LIN {X 61.321,Y 108.503,Z 73.500,A 180.000,B 0.000,C 180.000} C_DIS
LIN {X 61.500,Y 108.424,Z 73.500,A 180.000,B 0.000,C 180.000} C_DIS
LIN {X 61.692,Y 108.338,Z 73.500,A 180.000,B 0.000,C 180.000} C_DIS
LIN {X 61.858,Y 108.262,Z 73.500,A 180.000,B 0.000,C 180.000} C_DIS
LIN {X 62.036,Y 108.167,Z 73.500,A 180.000,B 0.000,C 180.000} C_DIS
LIN {X 62.371,Y 107.980,Z 73.500,A 180.000,B 0.000,C 180.000} C_DIS
LIN {X 62.394,Y 107.967,Z 73.500,A 180.000,B 0.000,C 180.000} C_DIS
LIN {X 62.573,Y 107.855,Z 73.500,A 180.000,B 0.000,C 180.000} C_DIS
LIN {X 62.930,Y 107.612,Z 73.500,A 180.000,B 0.000,C 180.000} C_DIS
LIN {X 63.020,Y 107.548,Z 73.500,A 180.000,B 0.000,C 180.000} C_DIS
LIN {X 63.109,Y 107.478,Z 73.500,A 180.000,B 0.000,C 180.000} C_DIS
LIN {X 63.369,Y 107.265,Z 73.500,A 180.000,B 0.000,C 180.000} C_DIS
LIN {X 63.467,Y 107.185,Z 73.500,A 180.000,B 0.000,C 180.000} C_DIS
LIN {X 63.578,Y 107.086,Z 73.500,A 180.000,B 0.000,C 180.000} C_DIS
LIN {X 63.645,Y 107.021,Z 73.500,A 180.000,B 0.000,C 180.000} C_DIS
LIN {X 63.824,Y 106.847,Z 73.500,A 180.000,B 0.000,C 180.000} C_DIS
LIN {X 63.944,Y 106.729,Z 73.500,A 180.000,B 0.000,C 180.000} C_DIS
LIN {X 64.003,Y 106.669,Z 73.500,A 180.000,B 0.000,C 180.000} C_DIS
LIN {X 64.109,Y 106.550,Z 73.500,A 180.000,B 0.000,C 180.000} C_DIS
LIN {X 64.360,Y 106.256,Z 73.500,A 180.000,B 0.000,C 180.000} C_DIS
LIN {X 64.414,Y 106.193,Z 73.500,A 180.000,B 0.000,C 180.000} C_DIS
LIN {X 64.539,Y 106.026,Z 73.500,A 180.000,B 0.000,C 180.000} C_DIS
LIN {X 64.718,Y 105.776,Z 73.500,A 180.000,B 0.000,C 180.000} C_DIS
LIN {X 64.802,Y 105.656,Z 73.500,A 180.000,B 0.000,C 180.000} C_DIS
LIN {X 64.897,Y 105.507,Z 73.500,A 180.000,B 0.000,C 180.000} C_DIS
LIN {X 65.075,Y 105.203,Z 73.500,A 180.000,B 0.000,C 180.000} C_DIS
LIN {X 65.124,Y 105.120,Z 73.500,A 180.000,B 0.000,C 180.000} C_DIS
LIN {X 65.219,Y 104.941,Z 73.500,A 180.000,B 0.000,C 180.000} C_DIS
LIN {X 65.254,Y 104.866,Z 73.500,A 180.000,B 0.000,C 180.000} C_DIS
LIN {X 65.388,Y 104.584,Z 73.500,A 180.000,B 0.000,C 180.000} C_DIS
LIN {X 65.433,Y 104.488,Z 73.500,A 180.000,B 0.000,C 180.000} C_DIS
LIN {X 65.469,Y 104.405,Z 73.500,A 180.000,B 0.000,C 180.000} C_DIS
LIN {X 65.536,Y 104.226,Z 73.500,A 180.000,B 0.000,C 180.000} C_DIS
LIN {X 65.612,Y 104.022,Z 73.500,A 180.000,B 0.000,C 180.000} C_DIS
LIN {X 65.668,Y 103.869,Z 73.500,A 180.000,B 0.000,C 180.000} C_DIS
LIN {X 65.724,Y 103.690,Z 73.500,A 180.000,B 0.000,C 180.000} C_DIS
LIN {X 65.821,Y 103.332,Z 73.500,A 180.000,B 0.000,C 180.000} C_DIS
LIN {X 65.867,Y 103.153,Z 73.500,A 180.000,B 0.000,C 180.000} C_DIS
LIN {X 65.901,Y 102.975,Z 73.500,A 180.000,B 0.000,C 180.000} C_DIS
LIN {X 65.965,Y 102.617,Z 73.500,A 180.000,B 0.000,C 180.000} C_DIS
LIN {X 65.969,Y 102.592,Z 73.500,A 180.000,B 0.000,C 180.000} C_DIS
LIN {X 65.991,Y 102.438,Z 73.500,A 180.000,B 0.000,C 180.000} C_DIS
LIN {X 66.007,Y 102.260,Z 73.500,A 180.000,B 0.000,C 180.000} C_DIS
LIN {X 66.023,Y 102.081,Z 73.500,A 180.000,B 0.000,C 180.000} C_DIS
LIN {X 66.039,Y 101.902,Z 73.500,A 180.000,B 0.000,C 180.000} C_DIS
LIN {X 66.045,Y 101.723,Z 73.500,A 180.000,B 0.000,C 180.000} C_DIS
LIN {X 66.045,Y 101.366,Z 73.500,A 180.000,B 0.000,C 180.000} C_DIS
LIN {X 66.043,Y 101.187,Z 73.500,A 180.000,B 0.000,C 180.000} C_DIS
LIN {X 66.031,Y 101.008,Z 73.500,A 180.000,B 0.000,C 180.000} C_DIS
LIN {X 65.999,Y 100.651,Z 73.500,A 180.000,B 0.000,C 180.000} C_DIS
LIN {X 65.980,Y 100.472,Z 73.500,A 180.000,B 0.000,C 180.000} C_DIS
LIN {X 65.969,Y 100.408,Z 73.500,A 180.000,B 0.000,C 180.000} C_DIS
LIN {X 65.949,Y 100.293,Z 73.500,A 180.000,B 0.000,C 180.000} C_DIS
LIN {X 65.917,Y 100.114,Z 73.500,A 180.000,B 0.000,C 180.000} C_DIS
LIN {X 65.885,Y 99.936,Z 73.500,A 180.000,B 0.000,C 180.000} C_DIS
LIN {X 65.845,Y 99.757,Z 73.500,A 180.000,B 0.000,C 180.000} C_DIS
LIN {X 65.796,Y 99.578,Z 73.500,A 180.000,B 0.000,C 180.000} C_DIS
LIN {X 65.748,Y 99.399,Z 73.500,A 180.000,B 0.000,C 180.000} C_DIS
LIN {X 65.698,Y 99.221,Z 73.500,A 180.000,B 0.000,C 180.000} C_DIS
LIN {X 65.635,Y 99.042,Z 73.500,A 180.000,B 0.000,C 180.000} C_DIS
LIN {X 65.503,Y 98.684,Z 73.500,A 180.000,B 0.000,C 180.000} C_DIS
LIN {X 65.433,Y 98.512,Z 73.500,A 180.000,B 0.000,C 180.000} C_DIS
LIN {X 65.430,Y 98.505,Z 73.500,A 180.000,B 0.000,C 180.000} C_DIS
LIN {X 65.346,Y 98.327,Z 73.500,A 180.000,B 0.000,C 180.000} C_DIS
LIN {X 65.254,Y 98.134,Z 73.500,A 180.000,B 0.000,C 180.000} C_DIS
LIN {X 65.174,Y 97.969,Z 73.500,A 180.000,B 0.000,C 180.000} C_DIS
LIN {X 65.075,Y 97.797,Z 73.500,A 180.000,B 0.000,C 180.000} C_DIS
LIN {X 64.897,Y 97.493,Z 73.500,A 180.000,B 0.000,C 180.000} C_DIS
LIN {X 64.861,Y 97.433,Z 73.500,A 180.000,B 0.000,C 180.000} C_DIS
LIN {X 64.739,Y 97.254,Z 73.500,A 180.000,B 0.000,C 180.000} C_DIS
LIN {X 64.539,Y 96.974,Z 73.500,A 180.000,B 0.000,C 180.000} C_DIS
LIN {X 64.484,Y 96.897,Z 73.500,A 180.000,B 0.000,C 180.000} C_DIS
LIN {X 64.360,Y 96.744,Z 73.500,A 180.000,B 0.000,C 180.000} C_DIS
LIN {X 64.182,Y 96.535,Z 73.500,A 180.000,B 0.000,C 180.000} C_DIS
LIN {X 64.030,Y 96.360,Z 73.500,A 180.000,B 0.000,C 180.000} C_DIS
LIN {X 64.003,Y 96.331,Z 73.500,A 180.000,B 0.000,C 180.000} C_DIS
LIN {X 63.853,Y 96.181,Z 73.500,A 180.000,B 0.000,C 180.000} C_DIS
LIN {X 63.645,Y 95.979,Z 73.500,A 180.000,B 0.000,C 180.000} C_DIS
LIN {X 63.477,Y 95.824,Z 73.500,A 180.000,B 0.000,C 180.000} C_DIS
LIN {X 63.467,Y 95.815,Z 73.500,A 180.000,B 0.000,C 180.000} C_DIS
LIN {X 63.288,Y 95.669,Z 73.500,A 180.000,B 0.000,C 180.000} C_DIS
LIN {X 63.109,Y 95.522,Z 73.500,A 180.000,B 0.000,C 180.000} C_DIS
LIN {X 63.038,Y 95.466,Z 73.500,A 180.000,B 0.000,C 180.000} C_DIS
LIN {X 62.930,Y 95.388,Z 73.500,A 180.000,B 0.000,C 180.000} C_DIS
LIN {X 62.573,Y 95.145,Z 73.500,A 180.000,B 0.000,C 180.000} C_DIS
LIN {X 62.518,Y 95.109,Z 73.500,A 180.000,B 0.000,C 180.000} C_DIS
LIN {X 62.394,Y 95.033,Z 73.500,A 180.000,B 0.000,C 180.000} C_DIS
LIN {X 62.210,Y 94.930,Z 73.500,A 180.000,B 0.000,C 180.000} C_DIS
LIN {X 62.036,Y 94.833,Z 73.500,A 180.000,B 0.000,C 180.000} C_DIS
LIN {X 61.885,Y 94.751,Z 73.500,A 180.000,B 0.000,C 180.000} C_DIS
LIN {X 61.858,Y 94.738,Z 73.500,A 180.000,B 0.000,C 180.000} C_DIS
LIN {X 61.679,Y 94.656,Z 73.500,A 180.000,B 0.000,C 180.000} C_DIS
LIN {X 61.491,Y 94.573,Z 73.500,A 180.000,B 0.000,C 180.000} C_DIS
LIN {X 61.321,Y 94.497,Z 73.500,A 180.000,B 0.000,C 180.000} C_DIS
LIN {X 61.143,Y 94.430,Z 73.500,A 180.000,B 0.000,C 180.000} C_DIS
LIN {X 60.785,Y 94.307,Z 73.500,A 180.000,B 0.000,C 180.000} C_DIS
LIN {X 60.606,Y 94.250,Z 73.500,A 180.000,B 0.000,C 180.000} C_DIS
LIN {X 60.470,Y 94.215,Z 73.500,A 180.000,B 0.000,C 180.000} C_DIS
LIN {X 60.249,Y 94.160,Z 73.500,A 180.000,B 0.000,C 180.000} C_DIS
LIN {X 60.070,Y 94.116,Z 73.500,A 180.000,B 0.000,C 180.000} C_DIS
LIN {X 59.891,Y 94.081,Z 73.500,A 180.000,B 0.000,C 180.000} C_DIS
LIN {X 59.534,Y 94.025,Z 73.500,A 180.000,B 0.000,C 180.000} C_DIS
LIN {X 59.355,Y 93.999,Z 73.500,A 180.000,B 0.000,C 180.000} C_DIS
LIN {X 59.176,Y 93.983,Z 73.500,A 180.000,B 0.000,C 180.000} C_DIS
LIN {X 58.819,Y 93.959,Z 73.500,A 180.000,B 0.000,C 180.000} C_DIS
LIN {X 58.640,Y 93.951,Z 73.500,A 180.000,B 0.000,C 180.000} C_DIS
LIN {X 58.461,Y 93.954,Z 73.500,A 180.000,B 0.000,C 180.000} C_DIS
LIN {X 58.103,Y 93.962,Z 73.500,A 180.000,B 0.000,C 180.000} C_DIS
LIN {X 57.925,Y 93.973,Z 73.500,A 180.000,B 0.000,C 180.000} C_DIS
LIN {X 57.746,Y 93.992,Z 73.500,A 180.000,B 0.000,C 180.000} C_DIS
LIN {X 57.567,Y 94.012,Z 73.500,A 180.000,B 0.000,C 180.000} C_DIS
LIN {X 57.388,Y 94.033,Z 73.500,A 180.000,B 0.000,C 180.000} C_DIS
LIN {X 57.363,Y 94.036,Z 73.500,A 180.000,B 0.000,C 180.000} C_DIS
LIN {X 57.210,Y 94.063,Z 73.500,A 180.000,B 0.000,C 180.000} C_DIS
LIN {X 56.852,Y 94.135,Z 73.500,A 180.000,B 0.000,C 180.000} C_DIS
LIN {X 56.673,Y 94.174,Z 73.500,A 180.000,B 0.000,C 180.000} C_DIS
LIN {X 56.528,Y 94.215,Z 73.500,A 180.000,B 0.000,C 180.000} C_DIS
LIN {X 56.316,Y 94.278,Z 73.500,A 180.000,B 0.000,C 180.000} C_DIS
LIN {X 56.137,Y 94.331,Z 73.500,A 180.000,B 0.000,C 180.000} C_DIS
LIN {X 55.958,Y 94.392,Z 73.500,A 180.000,B 0.000,C 180.000} C_DIS
LIN {X 55.953,Y 94.394,Z 73.500,A 180.000,B 0.000,C 180.000} C_DIS
LIN {X 55.779,Y 94.462,Z 73.500,A 180.000,B 0.000,C 180.000} C_DIS
LIN {X 55.601,Y 94.533,Z 73.500,A 180.000,B 0.000,C 180.000} C_DIS
LIN {X 55.501,Y 94.573,Z 73.500,A 180.000,B 0.000,C 180.000} C_DIS
LIN {X 55.422,Y 94.606,Z 73.500,A 180.000,B 0.000,C 180.000} C_DIS
LIN {X 55.243,Y 94.693,Z 73.500,A 180.000,B 0.000,C 180.000} C_DIS
LIN {X 55.064,Y 94.782,Z 73.500,A 180.000,B 0.000,C 180.000} C_DIS
LIN {X 54.886,Y 94.872,Z 73.500,A 180.000,B 0.000,C 180.000} C_DIS
LIN {X 54.781,Y 94.930,Z 73.500,A 180.000,B 0.000,C 180.000} C_DIS
LIN {X 54.707,Y 94.975,Z 73.500,A 180.000,B 0.000,C 180.000} C_DIS
LIN {X 54.349,Y 95.195,Z 73.500,A 180.000,B 0.000,C 180.000} C_DIS
LIN {X 54.210,Y 95.288,Z 73.500,A 180.000,B 0.000,C 180.000} C_DIS
LIN {X 54.171,Y 95.316,Z 73.500,A 180.000,B 0.000,C 180.000} C_DIS
LIN {X 53.970,Y 95.466,Z 73.500,A 180.000,B 0.000,C 180.000} C_DIS
LIN {X 53.813,Y 95.583,Z 73.500,A 180.000,B 0.000,C 180.000} C_DIS
LIN {X 53.733,Y 95.645,Z 73.500,A 180.000,B 0.000,C 180.000} C_DIS
LIN {X 53.634,Y 95.729,Z 73.500,A 180.000,B 0.000,C 180.000} C_DIS
LIN {X 53.329,Y 96.003,Z 73.500,A 180.000,B 0.000,C 180.000} C_DIS
LIN {X 53.277,Y 96.050,Z 73.500,A 180.000,B 0.000,C 180.000} C_DIS
LIN {X 53.144,Y 96.181,Z 73.500,A 180.000,B 0.000,C 180.000} C_DIS
LIN {X 52.919,Y 96.421,Z 73.500,A 180.000,B 0.000,C 180.000} C_DIS
LIN {X 52.810,Y 96.539,Z 73.500,A 180.000,B 0.000,C 180.000} C_DIS
LIN {X 52.740,Y 96.619,Z 73.500,A 180.000,B 0.000,C 180.000} C_DIS
LIN {X 52.662,Y 96.718,Z 73.500,A 180.000,B 0.000,C 180.000} C_DIS
LIN {X 52.522,Y 96.897,Z 73.500,A 180.000,B 0.000,C 180.000} C_DIS
LIN {X 52.383,Y 97.075,Z 73.500,A 180.000,B 0.000,C 180.000} C_DIS
LIN {X 52.261,Y 97.254,Z 73.500,A 180.000,B 0.000,C 180.000} C_DIS
LIN {X 52.145,Y 97.433,Z 73.500,A 180.000,B 0.000,C 180.000} C_DIS
LIN {X 52.029,Y 97.612,Z 73.500,A 180.000,B 0.000,C 180.000} C_DIS
LIN {X 52.025,Y 97.618,Z 73.500,A 180.000,B 0.000,C 180.000} C_DIS
LIN {X 51.927,Y 97.790,Z 73.500,A 180.000,B 0.000,C 180.000} C_DIS
LIN {X 51.737,Y 98.148,Z 73.500,A 180.000,B 0.000,C 180.000} C_DIS
LIN {X 51.668,Y 98.287,Z 73.500,A 180.000,B 0.000,C 180.000} C_DIS
LIN {X 51.650,Y 98.327,Z 73.500,A 180.000,B 0.000,C 180.000} C_DIS
LIN {X 51.574,Y 98.505,Z 73.500,A 180.000,B 0.000,C 180.000} C_DIS
LIN {X 51.489,Y 98.708,Z 73.500,A 180.000,B 0.000,C 180.000} C_DIS
LIN {X 51.426,Y 98.863,Z 73.500,A 180.000,B 0.000,C 180.000} C_DIS
LIN {X 51.365,Y 99.042,Z 73.500,A 180.000,B 0.000,C 180.000} C_DIS
LIN {X 51.250,Y 99.399,Z 73.500,A 180.000,B 0.000,C 180.000} C_DIS
LIN {X 51.199,Y 99.578,Z 73.500,A 180.000,B 0.000,C 180.000} C_DIS
LIN {X 51.159,Y 99.757,Z 73.500,A 180.000,B 0.000,C 180.000} C_DIS
LIN {X 51.118,Y 99.936,Z 73.500,A 180.000,B 0.000,C 180.000} C_DIS
LIN {X 51.079,Y 100.114,Z 73.500,A 180.000,B 0.000,C 180.000} C_DIS
LIN {X 51.049,Y 100.293,Z 73.500,A 180.000,B 0.000,C 180.000} C_DIS
LIN {X 51.001,Y 100.651,Z 73.500,A 180.000,B 0.000,C 180.000} C_DIS
LIN {X 50.980,Y 100.829,Z 73.500,A 180.000,B 0.000,C 180.000} C_DIS
LIN {X 50.969,Y 101.008,Z 73.500,A 180.000,B 0.000,C 180.000} C_DIS
LIN {X 50.953,Y 101.385,Z 73.500,A 180.000,B 0.000,C 180.000} C_DIS
LIN {X 50.950,Y 101.545,Z 73.500,A 180.000,B 0.000,C 180.000} C_DIS
LIN {X 50.953,Y 101.615,Z 73.500,A 180.000,B 0.000,C 180.000} C_DIS
LIN {X 50.965,Y 101.902,Z 73.500,A 180.000,B 0.000,C 180.000} C_DIS
LIN {X 50.973,Y 102.081,Z 73.500,A 180.000,B 0.000,C 180.000} C_DIS
LIN {X 50.989,Y 102.260,Z 73.500,A 180.000,B 0.000,C 180.000} C_DIS
LIN {X 51.013,Y 102.438,Z 73.500,A 180.000,B 0.000,C 180.000} C_DIS
LIN {X 51.037,Y 102.617,Z 73.500,A 180.000,B 0.000,C 180.000} C_DIS
LIN {X 51.062,Y 102.796,Z 73.500,A 180.000,B 0.000,C 180.000} C_DIS
LIN {X 51.098,Y 102.975,Z 73.500,A 180.000,B 0.000,C 180.000} C_DIS
LIN {X 51.179,Y 103.332,Z 73.500,A 180.000,B 0.000,C 180.000} C_DIS
LIN {X 51.223,Y 103.511,Z 73.500,A 180.000,B 0.000,C 180.000} C_DIS
LIN {X 51.279,Y 103.690,Z 73.500,A 180.000,B 0.000,C 180.000} C_DIS
LIN {X 51.336,Y 103.869,Z 73.500,A 180.000,B 0.000,C 180.000} C_DIS
LIN {X 51.393,Y 104.047,Z 73.500,A 180.000,B 0.000,C 180.000} C_DIS
LIN {X 51.461,Y 104.226,Z 73.500,A 180.000,B 0.000,C 180.000} C_DIS
LIN {X 51.612,Y 104.584,Z 73.500,A 180.000,B 0.000,C 180.000} C_DIS
LIN {X 51.668,Y 104.713,Z 73.500,A 180.000,B 0.000,C 180.000} C_DIS
LIN {X 51.691,Y 104.762,Z 73.500,A 180.000,B 0.000,C 180.000} C_DIS
LIN {X 51.785,Y 104.941,Z 73.500,A 180.000,B 0.000,C 180.000} C_DIS
LIN {X 51.879,Y 105.120,Z 73.500,A 180.000,B 0.000,C 180.000} C_DIS
LIN {X 51.975,Y 105.299,Z 73.500,A 180.000,B 0.000,C 180.000} C_DIS
LIN {X 52.025,Y 105.382,Z 73.500,A 180.000,B 0.000,C 180.000} C_DIS
LIN {X 52.087,Y 105.477,Z 73.500,A 180.000,B 0.000,C 180.000} C_DIS
LIN {X 52.204,Y 105.658,Z 73.500,A 180.000,B 0.000,C 180.000} C_DIS
LIN {X 52.319,Y 105.835,Z 73.500,A 180.000,B 0.000,C 180.000} C_DIS
LIN {X 52.383,Y 105.925,Z 73.500,A 180.000,B 0.000,C 180.000} C_DIS
LIN {X 52.452,Y 106.014,Z 73.500,A 180.000,B 0.000,C 180.000} C_DIS
LIN {X 52.591,Y 106.193,Z 73.500,A 180.000,B 0.000,C 180.000} C_DIS
LIN {X 52.732,Y 106.371,Z 73.500,A 180.000,B 0.000,C 180.000} C_DIS
LIN {X 52.740,Y 106.381,Z 73.500,A 180.000,B 0.000,C 180.000} C_DIS
LIN {X 52.892,Y 106.550,Z 73.500,A 180.000,B 0.000,C 180.000} C_DIS
LIN {X 53.098,Y 106.770,Z 73.500,A 180.000,B 0.000,C 180.000} C_DIS
LIN {X 53.231,Y 106.908,Z 73.500,A 180.000,B 0.000,C 180.000} C_DIS
LIN {X 53.277,Y 106.950,Z 73.500,A 180.000,B 0.000,C 180.000} C_DIS
LIN {X 53.428,Y 107.086,Z 73.500,A 180.000,B 0.000,C 180.000} C_DIS
LIN {X 53.634,Y 107.271,Z 73.500,A 180.000,B 0.000,C 180.000} C_DIS
LIN {X 53.724,Y 107.347,Z 73.500,A 180.000,B 0.000,C 180.000} C_DIS
LIN {X 53.813,Y 107.417,Z 73.500,A 180.000,B 0.000,C 180.000} C_DIS
LIN {X 54.089,Y 107.623,Z 73.500,A 180.000,B 0.000,C 180.000} C_DIS
LIN {X 54.171,Y 107.684,Z 73.500,A 180.000,B 0.000,C 180.000} C_DIS
LIN {X 54.344,Y 107.802,Z 73.500,A 180.000,B 0.000,C 180.000} C_DIS
LIN {X 54.707,Y 108.025,Z 73.500,A 180.000,B 0.000,C 180.000} C_DIS
LIN {X 54.886,Y 108.128,Z 73.500,A 180.000,B 0.000,C 180.000} C_DIS
LIN {X 54.947,Y 108.159,Z 73.500,A 180.000,B 0.000,C 180.000} C_DIS
LIN {X 55.304,Y 108.338,Z 73.500,A 180.000,B 0.000,C 180.000} C_DIS
LIN {X 55.422,Y 108.394,Z 73.500,A 180.000,B 0.000,C 180.000} C_DIS
LIN {X 55.601,Y 108.467,Z 73.500,A 180.000,B 0.000,C 180.000} C_DIS
LIN {X 55.779,Y 108.538,Z 73.500,A 180.000,B 0.000,C 180.000} C_DIS
LIN {X 55.958,Y 108.608,Z 73.500,A 180.000,B 0.000,C 180.000} C_DIS
LIN {X 56.137,Y 108.669,Z 73.500,A 180.000,B 0.000,C 180.000} C_DIS
LIN {X 56.225,Y 108.695,Z 73.500,A 180.000,B 0.000,C 180.000} C_DIS
LIN {X 56.495,Y 108.775,Z 73.500,A 180.000,B 0.000,C 180.000} C_DIS
LIN {X 56.673,Y 108.826,Z 73.500,A 180.000,B 0.000,C 180.000} C_DIS
LIN {X 56.852,Y 108.865,Z 73.500,A 180.000,B 0.000,C 180.000} C_DIS
LIN {X 57.210,Y 108.937,Z 73.500,A 180.000,B 0.000,C 180.000} C_DIS
LIN {X 57.388,Y 108.967,Z 73.500,A 180.000,B 0.000,C 180.000} C_DIS
LIN {X 57.567,Y 108.988,Z 73.500,A 180.000,B 0.000,C 180.000} C_DIS
LIN {X 57.746,Y 109.008,Z 73.500,A 180.000,B 0.000,C 180.000} C_DIS
LIN {X 57.925,Y 109.027,Z 73.500,A 180.000,B 0.000,C 180.000} C_DIS
LIN {X 58.103,Y 109.038,Z 73.500,A 180.000,B 0.000,C 180.000} C_DIS
LIN {X 58.461,Y 109.046,Z 73.500,A 180.000,B 0.000,C 180.000} C_DIS
LIN {X 58.640,Y 109.049,Z 73.500,A 180.000,B 0.000,C 180.000} C_DIS
LIN {X 58.819,Y 109.041,Z 73.500,A 180.000,B 0.000,C 180.000} C_DIS
LIN {X 59.176,Y 109.017,Z 73.500,A 180.000,B 0.000,C 180.000} C_DIS
LIN {X 59.355,Y 109.001,Z 73.500,A 180.000,B 0.000,C 180.000} C_DIS
LIN {X 59.534,Y 108.975,Z 73.500,A 180.000,B 0.000,C 180.000} C_DIS
LIN {X 59.891,Y 108.919,Z 73.500,A 180.000,B 0.000,C 180.000} C_DIS
LIN {X 60.070,Y 108.884,Z 73.500,A 180.000,B 0.000,C 180.000} C_DIS
LIN {X 60.111,Y 108.874,Z 73.500,A 180.000,B 0.000,C 180.000} C_DIS
LIN {X 60.427,Y 108.796,Z 73.500,A 180.000,B 0.000,C 180.000} C_DIS
LIN {X 60.606,Y 108.750,Z 73.500,A 180.000,B 0.000,C 180.000} C_DIS
LIN {X 60.778,Y 108.695,Z 73.500,A 180.000,B 0.000,C 180.000} C_DIS
LIN {X 60.958,Y 108.633,Z 73.500,A 180.000,B 0.000,C 180.000} C_DIS
; Link Move Starts
LIN {X 61.255,Y 108.529,Z 73.500,A 180.000,B 0.000,C 180.000} C_DIS
LIN {X 61.544,Y 108.404,Z 73.499,A 180.000,B 0.000,C 180.000} C_DIS
LIN {X 61.831,Y 108.275,Z 73.498,A 180.000,B 0.000,C 180.000} C_DIS
LIN {X 62.109,Y 108.126,Z 73.496,A 180.000,B 0.000,C 180.000} C_DIS
LIN {X 62.384,Y 107.973,Z 73.494,A 180.000,B 0.000,C 180.000} C_DIS
LIN {X 62.649,Y 107.803,Z 73.491,A 180.000,B 0.000,C 180.000} C_DIS
LIN {X 62.910,Y 107.626,Z 73.488,A 180.000,B 0.000,C 180.000} C_DIS
LIN {X 63.038,Y 107.534,Z 73.487,A 180.000,B 0.000,C 180.000} C_DIS
LIN {X 63.161,Y 107.435,Z 73.485,A 180.000,B 0.000,C 180.000} C_DIS
LIN {X 63.404,Y 107.236,Z 73.481,A 180.000,B 0.000,C 180.000} C_DIS
LIN {X 63.525,Y 107.135,Z 73.479,A 180.000,B 0.000,C 180.000} C_DIS
LIN {X 63.640,Y 107.027,Z 73.477,A 180.000,B 0.000,C 180.000} C_DIS
LIN {X 63.865,Y 106.807,Z 73.472,A 180.000,B 0.000,C 180.000} C_DIS
LIN {X 63.977,Y 106.696,Z 73.469,A 180.000,B 0.000,C 180.000} C_DIS
LIN {X 64.084,Y 106.580,Z 73.467,A 180.000,B 0.000,C 180.000} C_DIS
LIN {X 64.186,Y 106.460,Z 73.464,A 180.000,B 0.000,C 180.000} C_DIS
LIN {X 64.288,Y 106.340,Z 73.461,A 180.000,B 0.000,C 180.000} C_DIS
LIN {X 64.391,Y 106.221,Z 73.459,A 180.000,B 0.000,C 180.000} C_DIS
LIN {X 64.488,Y 106.097,Z 73.456,A 180.000,B 0.000,C 180.000} C_DIS
LIN {X 64.580,Y 105.969,Z 73.452,A 180.000,B 0.000,C 180.000} C_DIS
LIN {X 64.672,Y 105.841,Z 73.449,A 180.000,B 0.000,C 180.000} C_DIS
LIN {X 64.763,Y 105.713,Z 73.446,A 180.000,B 0.000,C 180.000} C_DIS
LIN {X 64.851,Y 105.582,Z 73.443,A 180.000,B 0.000,C 180.000} C_DIS
LIN {X 64.932,Y 105.447,Z 73.439,A 180.000,B 0.000,C 180.000} C_DIS
LIN {X 65.012,Y 105.311,Z 73.436,A 180.000,B 0.000,C 180.000} C_DIS
LIN {X 65.092,Y 105.175,Z 73.432,A 180.000,B 0.000,C 180.000} C_DIS
LIN {X 65.169,Y 105.038,Z 73.428,A 180.000,B 0.000,C 180.000} C_DIS
LIN {X 65.239,Y 104.897,Z 73.425,A 180.000,B 0.000,C 180.000} C_DIS
LIN {X 65.307,Y 104.755,Z 73.421,A 180.000,B 0.000,C 180.000} C_DIS
LIN {X 65.374,Y 104.613,Z 73.417,A 180.000,B 0.000,C 180.000} C_DIS
LIN {X 65.441,Y 104.470,Z 73.413,A 180.000,B 0.000,C 180.000} C_DIS
LIN {X 65.500,Y 104.324,Z 73.409,A 180.000,B 0.000,C 180.000} C_DIS
LIN {X 65.555,Y 104.176,Z 73.405,A 180.000,B 0.000,C 180.000} C_DIS
LIN {X 65.609,Y 104.029,Z 73.400,A 180.000,B 0.000,C 180.000} C_DIS
LIN {X 65.664,Y 103.881,Z 73.396,A 180.000,B 0.000,C 180.000} C_DIS
LIN {X 65.712,Y 103.731,Z 73.392,A 180.000,B 0.000,C 180.000} C_DIS
LIN {X 65.754,Y 103.579,Z 73.387,A 180.000,B 0.000,C 180.000} C_DIS
LIN {X 65.795,Y 103.427,Z 73.383,A 180.000,B 0.000,C 180.000} C_DIS
LIN {X 65.836,Y 103.275,Z 73.378,A 180.000,B 0.000,C 180.000} C_DIS
LIN {X 65.874,Y 103.122,Z 73.373,A 180.000,B 0.000,C 180.000} C_DIS
LIN {X 65.902,Y 102.967,Z 73.369,A 180.000,B 0.000,C 180.000} C_DIS
LIN {X 65.930,Y 102.812,Z 73.364,A 180.000,B 0.000,C 180.000} C_DIS
LIN {X 65.958,Y 102.657,Z 73.359,A 180.000,B 0.000,C 180.000} C_DIS
LIN {X 65.983,Y 102.502,Z 73.354,A 180.000,B 0.000,C 180.000} C_DIS
LIN {X 65.993,Y 102.423,Z 73.351,A 180.000,B 0.000,C 180.000} C_DIS
LIN {X 66.000,Y 102.345,Z 73.349,A 180.000,B 0.000,C 180.000} C_DIS
LIN {X 66.007,Y 102.267,Z 73.346,A 180.000,B 0.000,C 180.000} C_DIS
LIN {X 66.014,Y 102.188,Z 73.344,A 180.000,B 0.000,C 180.000} C_DIS
LIN {X 66.021,Y 102.110,Z 73.341,A 180.000,B 0.000,C 180.000} C_DIS
LIN {X 66.028,Y 102.031,Z 73.339,A 180.000,B 0.000,C 180.000} C_DIS
LIN {X 66.035,Y 101.953,Z 73.336,A 180.000,B 0.000,C 180.000} C_DIS
LIN {X 66.040,Y 101.874,Z 73.333,A 180.000,B 0.000,C 180.000} C_DIS
LIN {X 66.044,Y 101.796,Z 73.331,A 180.000,B 0.000,C 180.000} C_DIS
LIN {X 66.045,Y 101.717,Z 73.328,A 180.000,B 0.000,C 180.000} C_DIS
LIN {X 66.045,Y 101.559,Z 73.323,A 180.000,B 0.000,C 180.000} C_DIS
LIN {X 66.045,Y 101.402,Z 73.317,A 180.000,B 0.000,C 180.000} C_DIS
LIN {X 66.045,Y 101.323,Z 73.315,A 180.000,B 0.000,C 180.000} C_DIS
LIN {X 66.045,Y 101.244,Z 73.312,A 180.000,B 0.000,C 180.000} C_DIS
LIN {X 66.043,Y 101.166,Z 73.309,A 180.000,B 0.000,C 180.000} C_DIS
LIN {X 66.038,Y 101.087,Z 73.307,A 180.000,B 0.000,C 180.000} C_DIS
LIN {X 66.031,Y 101.008,Z 73.304,A 180.000,B 0.000,C 180.000} C_DIS
LIN {X 66.017,Y 100.852,Z 73.298,A 180.000,B 0.000,C 180.000} C_DIS
LIN {X 66.010,Y 100.773,Z 73.296,A 180.000,B 0.000,C 180.000} C_DIS
LIN {X 65.996,Y 100.616,Z 73.290,A 180.000,B 0.000,C 180.000} C_DIS
LIN {X 65.988,Y 100.538,Z 73.287,A 180.000,B 0.000,C 180.000} C_DIS
LIN {X 65.978,Y 100.460,Z 73.285,A 180.000,B 0.000,C 180.000} C_DIS
LIN {X 65.965,Y 100.382,Z 73.282,A 180.000,B 0.000,C 180.000} C_DIS
LIN {X 65.937,Y 100.227,Z 73.276,A 180.000,B 0.000,C 180.000} C_DIS
LIN {X 65.923,Y 100.150,Z 73.274,A 180.000,B 0.000,C 180.000} C_DIS
LIN {X 65.896,Y 99.995,Z 73.268,A 180.000,B 0.000,C 180.000} C_DIS
LIN {X 65.881,Y 99.917,Z 73.265,A 180.000,B 0.000,C 180.000} C_DIS
LIN {X 65.865,Y 99.840,Z 73.263,A 180.000,B 0.000,C 180.000} C_DIS
LIN {X 65.847,Y 99.763,Z 73.260,A 180.000,B 0.000,C 180.000} C_DIS
LIN {X 65.826,Y 99.687,Z 73.257,A 180.000,B 0.000,C 180.000} C_DIS
LIN {X 65.764,Y 99.459,Z 73.249,A 180.000,B 0.000,C 180.000} C_DIS
LIN {X 65.723,Y 99.307,Z 73.243,A 180.000,B 0.000,C 180.000} C_DIS
LIN {X 65.701,Y 99.232,Z 73.241,A 180.000,B 0.000,C 180.000} C_DIS
LIN {X 65.677,Y 99.157,Z 73.238,A 180.000,B 0.000,C 180.000} C_DIS
LIN {X 65.650,Y 99.083,Z 73.235,A 180.000,B 0.000,C 180.000} C_DIS
LIN {X 65.514,Y 98.713,Z 73.221,A 180.000,B 0.000,C 180.000} C_DIS
LIN {X 65.486,Y 98.640,Z 73.219,A 180.000,B 0.000,C 180.000} C_DIS
LIN {X 65.457,Y 98.567,Z 73.216,A 180.000,B 0.000,C 180.000} C_DIS
LIN {X 65.425,Y 98.494,Z 73.213,A 180.000,B 0.000,C 180.000} C_DIS
LIN {X 65.391,Y 98.423,Z 73.210,A 180.000,B 0.000,C 180.000} C_DIS
LIN {X 65.358,Y 98.352,Z 73.208,A 180.000,B 0.000,C 180.000} C_DIS
LIN {X 65.290,Y 98.210,Z 73.202,A 180.000,B 0.000,C 180.000} C_DIS
LIN {X 65.223,Y 98.067,Z 73.197,A 180.000,B 0.000,C 180.000} C_DIS
LIN {X 65.188,Y 97.997,Z 73.194,A 180.000,B 0.000,C 180.000} C_DIS
LIN {X 65.151,Y 97.927,Z 73.191,A 180.000,B 0.000,C 180.000} C_DIS
LIN {X 65.112,Y 97.859,Z 73.188,A 180.000,B 0.000,C 180.000} C_DIS
LIN {X 65.072,Y 97.791,Z 73.186,A 180.000,B 0.000,C 180.000} C_DIS
LIN {X 64.992,Y 97.655,Z 73.180,A 180.000,B 0.000,C 180.000} C_DIS
LIN {X 64.912,Y 97.519,Z 73.175,A 180.000,B 0.000,C 180.000} C_DIS
LIN {X 64.872,Y 97.452,Z 73.172,A 180.000,B 0.000,C 180.000} C_DIS
LIN {X 64.830,Y 97.385,Z 73.169,A 180.000,B 0.000,C 180.000} C_DIS
LIN {X 64.786,Y 97.320,Z 73.166,A 180.000,B 0.000,C 180.000} C_DIS
LIN {X 64.740,Y 97.256,Z 73.164,A 180.000,B 0.000,C 180.000} C_DIS
LIN {X 64.603,Y 97.063,Z 73.155,A 180.000,B 0.000,C 180.000} C_DIS
LIN {X 64.512,Y 96.935,Z 73.150,A 180.000,B 0.000,C 180.000} C_DIS
LIN {X 64.465,Y 96.872,Z 73.147,A 180.000,B 0.000,C 180.000} C_DIS
LIN {X 64.416,Y 96.810,Z 73.144,A 180.000,B 0.000,C 180.000} C_DIS
LIN {X 64.365,Y 96.750,Z 73.142,A 180.000,B 0.000,C 180.000} C_DIS
LIN {X 64.212,Y 96.570,Z 73.133,A 180.000,B 0.000,C 180.000} C_DIS
LIN {X 64.109,Y 96.450,Z 73.128,A 180.000,B 0.000,C 180.000} C_DIS
LIN {X 64.058,Y 96.391,Z 73.125,A 180.000,B 0.000,C 180.000} C_DIS
LIN {X 64.005,Y 96.333,Z 73.122,A 180.000,B 0.000,C 180.000} C_DIS
LIN {X 63.950,Y 96.276,Z 73.120,A 180.000,B 0.000,C 180.000} C_DIS
LIN {X 63.894,Y 96.221,Z 73.117,A 180.000,B 0.000,C 180.000} C_DIS
LIN {X 63.612,Y 95.946,Z 73.103,A 180.000,B 0.000,C 180.000} C_DIS
LIN {X 63.555,Y 95.892,Z 73.100,A 180.000,B 0.000,C 180.000} C_DIS
LIN {X 63.496,Y 95.840,Z 73.098,A 180.000,B 0.000,C 180.000} C_DIS
LIN {X 63.435,Y 95.789,Z 73.095,A 180.000,B 0.000,C 180.000} C_DIS
LIN {X 63.131,Y 95.540,Z 73.081,A 180.000,B 0.000,C 180.000} C_DIS
LIN {X 63.069,Y 95.490,Z 73.078,A 180.000,B 0.000,C 180.000} C_DIS
LIN {X 63.007,Y 95.443,Z 73.076,A 180.000,B 0.000,C 180.000} C_DIS
LIN {X 62.943,Y 95.397,Z 73.073,A 180.000,B 0.000,C 180.000} C_DIS
LIN {X 62.877,Y 95.353,Z 73.070,A 180.000,B 0.000,C 180.000} C_DIS
LIN {X 62.617,Y 95.175,Z 73.059,A 180.000,B 0.000,C 180.000} C_DIS
LIN {X 62.552,Y 95.131,Z 73.056,A 180.000,B 0.000,C 180.000} C_DIS
LIN {X 62.486,Y 95.088,Z 73.054,A 180.000,B 0.000,C 180.000} C_DIS
LIN {X 62.419,Y 95.047,Z 73.051,A 180.000,B 0.000,C 180.000} C_DIS
LIN {X 62.350,Y 95.008,Z 73.048,A 180.000,B 0.000,C 180.000} C_DIS
LIN {X 62.006,Y 94.816,Z 73.034,A 180.000,B 0.000,C 180.000} C_DIS
LIN {X 61.937,Y 94.778,Z 73.032,A 180.000,B 0.000,C 180.000} C_DIS
LIN {X 61.867,Y 94.743,Z 73.029,A 180.000,B 0.000,C 180.000} C_DIS
LIN {X 61.796,Y 94.709,Z 73.026,A 180.000,B 0.000,C 180.000} C_DIS
LIN {X 61.724,Y 94.677,Z 73.023,A 180.000,B 0.000,C 180.000} C_DIS
LIN {X 61.437,Y 94.548,Z 73.012,A 180.000,B 0.000,C 180.000} C_DIS
LIN {X 61.365,Y 94.516,Z 73.010,A 180.000,B 0.000,C 180.000} C_DIS
LIN {X 61.292,Y 94.485,Z 73.007,A 180.000,B 0.000,C 180.000} C_DIS
LIN {X 61.219,Y 94.457,Z 73.004,A 180.000,B 0.000,C 180.000} C_DIS
LIN {X 61.144,Y 94.431,Z 73.001,A 180.000,B 0.000,C 180.000} C_DIS
LIN {X 60.772,Y 94.302,Z 72.988,A 180.000,B 0.000,C 180.000} C_DIS
LIN {X 60.697,Y 94.277,Z 72.985,A 180.000,B 0.000,C 180.000} C_DIS
LIN {X 60.622,Y 94.254,Z 72.982,A 180.000,B 0.000,C 180.000} C_DIS
LIN {X 60.546,Y 94.234,Z 72.979,A 180.000,B 0.000,C 180.000} C_DIS
LIN {X 60.470,Y 94.215,Z 72.977,A 180.000,B 0.000,C 180.000} C_DIS
LIN {X 60.164,Y 94.139,Z 72.966,A 180.000,B 0.000,C 180.000} C_DIS
LIN {X 60.088,Y 94.120,Z 72.963,A 180.000,B 0.000,C 180.000} C_DIS
LIN {X 60.011,Y 94.103,Z 72.960,A 180.000,B 0.000,C 180.000} C_DIS
LIN {X 59.933,Y 94.088,Z 72.957,A 180.000,B 0.000,C 180.000} C_DIS
LIN {X 59.856,Y 94.075,Z 72.955,A 180.000,B 0.000,C 180.000} C_DIS
LIN {X 59.467,Y 94.014,Z 72.941,A 180.000,B 0.000,C 180.000} C_DIS
LIN {X 59.389,Y 94.003,Z 72.938,A 180.000,B 0.000,C 180.000} C_DIS
LIN {X 59.310,Y 93.994,Z 72.935,A 180.000,B 0.000,C 180.000} C_DIS
LIN {X 59.232,Y 93.987,Z 72.933,A 180.000,B 0.000,C 180.000} C_DIS
LIN {X 59.153,Y 93.982,Z 72.930,A 180.000,B 0.000,C 180.000} C_DIS
LIN {X 58.839,Y 93.961,Z 72.919,A 180.000,B 0.000,C 180.000} C_DIS
LIN {X 58.761,Y 93.956,Z 72.916,A 180.000,B 0.000,C 180.000} C_DIS
LIN {X 58.682,Y 93.952,Z 72.913,A 180.000,B 0.000,C 180.000} C_DIS
LIN {X 58.603,Y 93.951,Z 72.911,A 180.000,B 0.000,C 180.000} C_DIS
LIN {X 58.524,Y 93.953,Z 72.908,A 180.000,B 0.000,C 180.000} C_DIS
LIN {X 58.131,Y 93.961,Z 72.894,A 180.000,B 0.000,C 180.000} C_DIS
LIN {X 58.052,Y 93.964,Z 72.891,A 180.000,B 0.000,C 180.000} C_DIS
LIN {X 57.973,Y 93.968,Z 72.889,A 180.000,B 0.000,C 180.000} C_DIS
LIN {X 57.895,Y 93.976,Z 72.886,A 180.000,B 0.000,C 180.000} C_DIS
LIN {X 57.738,Y 93.993,Z 72.880,A 180.000,B 0.000,C 180.000} C_DIS
LIN {X 57.582,Y 94.011,Z 72.875,A 180.000,B 0.000,C 180.000} C_DIS
LIN {X 57.504,Y 94.019,Z 72.872,A 180.000,B 0.000,C 180.000} C_DIS
LIN {X 57.425,Y 94.028,Z 72.869,A 180.000,B 0.000,C 180.000} C_DIS
LIN {X 57.347,Y 94.039,Z 72.867,A 180.000,B 0.000,C 180.000} C_DIS
LIN {X 57.270,Y 94.052,Z 72.864,A 180.000,B 0.000,C 180.000} C_DIS
LIN {X 57.192,Y 94.067,Z 72.861,A 180.000,B 0.000,C 180.000} C_DIS
LIN {X 56.806,Y 94.145,Z 72.847,A 180.000,B 0.000,C 180.000} C_DIS
LIN {X 56.729,Y 94.161,Z 72.845,A 180.000,B 0.000,C 180.000} C_DIS
LIN {X 56.653,Y 94.180,Z 72.842,A 180.000,B 0.000,C 180.000} C_DIS
LIN {X 56.577,Y 94.201,Z 72.839,A 180.000,B 0.000,C 180.000} C_DIS
LIN {X 56.199,Y 94.312,Z 72.825,A 180.000,B 0.000,C 180.000} C_DIS
LIN {X 56.124,Y 94.335,Z 72.823,A 180.000,B 0.000,C 180.000} C_DIS
LIN {X 56.049,Y 94.359,Z 72.820,A 180.000,B 0.000,C 180.000} C_DIS
LIN {X 55.975,Y 94.386,Z 72.817,A 180.000,B 0.000,C 180.000} C_DIS
LIN {X 55.901,Y 94.414,Z 72.814,A 180.000,B 0.000,C 180.000} C_DIS
LIN {X 55.828,Y 94.443,Z 72.812,A 180.000,B 0.000,C 180.000} C_DIS
LIN {X 55.682,Y 94.501,Z 72.806,A 180.000,B 0.000,C 180.000} C_DIS
LIN {X 55.535,Y 94.559,Z 72.801,A 180.000,B 0.000,C 180.000} C_DIS
LIN {X 55.462,Y 94.588,Z 72.798,A 180.000,B 0.000,C 180.000} C_DIS
LIN {X 55.390,Y 94.620,Z 72.795,A 180.000,B 0.000,C 180.000} C_DIS
LIN {X 55.319,Y 94.655,Z 72.792,A 180.000,B 0.000,C 180.000} C_DIS
LIN {X 55.249,Y 94.690,Z 72.790,A 180.000,B 0.000,C 180.000} C_DIS
LIN {X 55.108,Y 94.760,Z 72.784,A 180.000,B 0.000,C 180.000} C_DIS
LIN {X 54.967,Y 94.831,Z 72.779,A 180.000,B 0.000,C 180.000} C_DIS
LIN {X 54.897,Y 94.866,Z 72.776,A 180.000,B 0.000,C 180.000} C_DIS
LIN {X 54.827,Y 94.903,Z 72.773,A 180.000,B 0.000,C 180.000} C_DIS
LIN {X 54.759,Y 94.943,Z 72.770,A 180.000,B 0.000,C 180.000} C_DIS
LIN {X 54.692,Y 94.984,Z 72.768,A 180.000,B 0.000,C 180.000} C_DIS
LIN {X 54.558,Y 95.067,Z 72.762,A 180.000,B 0.000,C 180.000} C_DIS
LIN {X 54.357,Y 95.191,Z 72.754,A 180.000,B 0.000,C 180.000} C_DIS
LIN {X 54.290,Y 95.233,Z 72.751,A 180.000,B 0.000,C 180.000} C_DIS
LIN {X 54.225,Y 95.277,Z 72.748,A 180.000,B 0.000,C 180.000} C_DIS
LIN {X 54.161,Y 95.323,Z 72.746,A 180.000,B 0.000,C 180.000} C_DIS
LIN {X 54.035,Y 95.417,Z 72.740,A 180.000,B 0.000,C 180.000} C_DIS
LIN {X 53.846,Y 95.559,Z 72.732,A 180.000,B 0.000,C 180.000} C_DIS
LIN {X 53.783,Y 95.606,Z 72.729,A 180.000,B 0.000,C 180.000} C_DIS
LIN {X 53.721,Y 95.655,Z 72.726,A 180.000,B 0.000,C 180.000} C_DIS
LIN {X 53.661,Y 95.706,Z 72.724,A 180.000,B 0.000,C 180.000} C_DIS
LIN {X 53.602,Y 95.758,Z 72.721,A 180.000,B 0.000,C 180.000} C_DIS
LIN {X 53.485,Y 95.863,Z 72.715,A 180.000,B 0.000,C 180.000} C_DIS
LIN {X 53.426,Y 95.916,Z 72.713,A 180.000,B 0.000,C 180.000} C_DIS
LIN {X 53.309,Y 96.021,Z 72.707,A 180.000,B 0.000,C 180.000} C_DIS
LIN {X 53.251,Y 96.074,Z 72.704,A 180.000,B 0.000,C 180.000} C_DIS
LIN {X 53.194,Y 96.129,Z 72.702,A 180.000,B 0.000,C 180.000} C_DIS
LIN {X 53.140,Y 96.186,Z 72.699,A 180.000,B 0.000,C 180.000} C_DIS
LIN {X 53.032,Y 96.301,Z 72.693,A 180.000,B 0.000,C 180.000} C_DIS
LIN {X 52.871,Y 96.473,Z 72.685,A 180.000,B 0.000,C 180.000} C_DIS
LIN {X 52.817,Y 96.531,Z 72.682,A 180.000,B 0.000,C 180.000} C_DIS
LIN {X 52.765,Y 96.590,Z 72.680,A 180.000,B 0.000,C 180.000} C_DIS
LIN {X 52.715,Y 96.650,Z 72.677,A 180.000,B 0.000,C 180.000} C_DIS
LIN {X 52.666,Y 96.712,Z 72.674,A 180.000,B 0.000,C 180.000} C_DIS
LIN {X 52.569,Y 96.836,Z 72.669,A 180.000,B 0.000,C 180.000} C_DIS
LIN {X 52.472,Y 96.960,Z 72.664,A 180.000,B 0.000,C 180.000} C_DIS
LIN {X 52.423,Y 97.022,Z 72.661,A 180.000,B 0.000,C 180.000} C_DIS
LIN {X 52.376,Y 97.085,Z 72.659,A 180.000,B 0.000,C 180.000} C_DIS
LIN {X 52.330,Y 97.149,Z 72.656,A 180.000,B 0.000,C 180.000} C_DIS
LIN {X 52.286,Y 97.215,Z 72.654,A 180.000,B 0.000,C 180.000} C_DIS
LIN {X 52.243,Y 97.281,Z 72.651,A 180.000,B 0.000,C 180.000} C_DIS
LIN {X 52.201,Y 97.347,Z 72.649,A 180.000,B 0.000,C 180.000} C_DIS
LIN {X 52.115,Y 97.479,Z 72.644,A 180.000,B 0.000,C 180.000} C_DIS
LIN {X 52.029,Y 97.611,Z 72.639,A 180.000,B 0.000,C 180.000} C_DIS
LIN {X 51.950,Y 97.747,Z 72.634,A 180.000,B 0.000,C 180.000} C_DIS
LIN {X 51.876,Y 97.886,Z 72.629,A 180.000,B 0.000,C 180.000} C_DIS
LIN {X 51.802,Y 98.026,Z 72.624,A 180.000,B 0.000,C 180.000} C_DIS
LIN {X 51.729,Y 98.165,Z 72.620,A 180.000,B 0.000,C 180.000} C_DIS
LIN {X 51.659,Y 98.306,Z 72.615,A 180.000,B 0.000,C 180.000} C_DIS
LIN {X 51.597,Y 98.451,Z 72.611,A 180.000,B 0.000,C 180.000} C_DIS
LIN {X 51.536,Y 98.596,Z 72.606,A 180.000,B 0.000,C 180.000} C_DIS
LIN {X 51.475,Y 98.741,Z 72.602,A 180.000,B 0.000,C 180.000} C_DIS
LIN {X 51.416,Y 98.888,Z 72.597,A 180.000,B 0.000,C 180.000} C_DIS
LIN {X 51.366,Y 99.037,Z 72.593,A 180.000,B 0.000,C 180.000} C_DIS
LIN {X 51.318,Y 99.187,Z 72.589,A 180.000,B 0.000,C 180.000} C_DIS
LIN {X 51.270,Y 99.337,Z 72.585,A 180.000,B 0.000,C 180.000} C_DIS
LIN {X 51.223,Y 99.487,Z 72.581,A 180.000,B 0.000,C 180.000} C_DIS
LIN {X 51.185,Y 99.640,Z 72.577,A 180.000,B 0.000,C 180.000} C_DIS
LIN {X 51.150,Y 99.794,Z 72.573,A 180.000,B 0.000,C 180.000} C_DIS
LIN {X 51.116,Y 99.947,Z 72.570,A 180.000,B 0.000,C 180.000} C_DIS
LIN {X 51.081,Y 100.101,Z 72.566,A 180.000,B 0.000,C 180.000} C_DIS
LIN {X 51.054,Y 100.256,Z 72.562,A 180.000,B 0.000,C 180.000} C_DIS
LIN {X 51.033,Y 100.412,Z 72.559,A 180.000,B 0.000,C 180.000} C_DIS
LIN {X 51.012,Y 100.568,Z 72.556,A 180.000,B 0.000,C 180.000} C_DIS
LIN {X 50.992,Y 100.724,Z 72.552,A 180.000,B 0.000,C 180.000} C_DIS
LIN {X 50.976,Y 100.881,Z 72.549,A 180.000,B 0.000,C 180.000} C_DIS
LIN {X 50.968,Y 101.038,Z 72.546,A 180.000,B 0.000,C 180.000} C_DIS
LIN {X 50.961,Y 101.196,Z 72.543,A 180.000,B 0.000,C 180.000} C_DIS
LIN {X 50.954,Y 101.353,Z 72.540,A 180.000,B 0.000,C 180.000} C_DIS
LIN {X 50.950,Y 101.511,Z 72.537,A 180.000,B 0.000,C 180.000} C_DIS
LIN {X 50.955,Y 101.668,Z 72.534,A 180.000,B 0.000,C 180.000} C_DIS
LIN {X 50.962,Y 101.825,Z 72.532,A 180.000,B 0.000,C 180.000} C_DIS
LIN {X 50.969,Y 101.983,Z 72.529,A 180.000,B 0.000,C 180.000} C_DIS
LIN {X 50.977,Y 102.140,Z 72.527,A 180.000,B 0.000,C 180.000} C_DIS
LIN {X 51.015,Y 102.453,Z 72.522,A 180.000,B 0.000,C 180.000} C_DIS
LIN {X 51.057,Y 102.765,Z 72.518,A 180.000,B 0.000,C 180.000} C_DIS
LIN {X 51.120,Y 103.073,Z 72.514,A 180.000,B 0.000,C 180.000} C_DIS
LIN {X 51.189,Y 103.381,Z 72.511,A 180.000,B 0.000,C 180.000} C_DIS
LIN {X 51.277,Y 103.683,Z 72.508,A 180.000,B 0.000,C 180.000} C_DIS
LIN {X 51.373,Y 103.983,Z 72.505,A 180.000,B 0.000,C 180.000} C_DIS
LIN {X 51.424,Y 104.132,Z 72.504,A 180.000,B 0.000,C 180.000} C_DIS
LIN {X 51.483,Y 104.278,Z 72.503,A 180.000,B 0.000,C 180.000} C_DIS
LIN {X 51.605,Y 104.569,Z 72.502,A 180.000,B 0.000,C 180.000} C_DIS
LIN {X 51.668,Y 104.713,Z 72.501,A 180.000,B 0.000,C 180.000} C_DIS
LIN {X 51.738,Y 104.854,Z 72.501,A 180.000,B 0.000,C 180.000} C_DIS
LIN {X 51.886,Y 105.132,Z 72.500,A 180.000,B 0.000,C 180.000} C_DIS
LIN {X 51.998,Y 105.336,Z 72.500,A 180.000,B 0.000,C 180.000} C_DIS
; Cutting Move Starts
LIN {X 52.025,Y 105.382,Z 72.500,A 180.000,B 0.000,C 180.000} C_DIS
LIN {X 52.087,Y 105.477,Z 72.500,A 180.000,B 0.000,C 180.000} C_DIS
LIN {X 52.204,Y 105.658,Z 72.500,A 180.000,B 0.000,C 180.000} C_DIS
LIN {X 52.319,Y 105.835,Z 72.500,A 180.000,B 0.000,C 180.000} C_DIS
LIN {X 52.383,Y 105.925,Z 72.500,A 180.000,B 0.000,C 180.000} C_DIS
LIN {X 52.452,Y 106.014,Z 72.500,A 180.000,B 0.000,C 180.000} C_DIS
LIN {X 52.591,Y 106.193,Z 72.500,A 180.000,B 0.000,C 180.000} C_DIS
LIN {X 52.732,Y 106.371,Z 72.500,A 180.000,B 0.000,C 180.000} C_DIS
LIN {X 52.740,Y 106.381,Z 72.500,A 180.000,B 0.000,C 180.000} C_DIS
LIN {X 52.892,Y 106.550,Z 72.500,A 180.000,B 0.000,C 180.000} C_DIS
LIN {X 53.098,Y 106.770,Z 72.500,A 180.000,B 0.000,C 180.000} C_DIS
LIN {X 53.231,Y 106.908,Z 72.500,A 180.000,B 0.000,C 180.000} C_DIS
LIN {X 53.277,Y 106.950,Z 72.500,A 180.000,B 0.000,C 180.000} C_DIS
LIN {X 53.428,Y 107.086,Z 72.500,A 180.000,B 0.000,C 180.000} C_DIS
LIN {X 53.634,Y 107.271,Z 72.500,A 180.000,B 0.000,C 180.000} C_DIS
LIN {X 53.724,Y 107.347,Z 72.500,A 180.000,B 0.000,C 180.000} C_DIS
LIN {X 53.813,Y 107.417,Z 72.500,A 180.000,B 0.000,C 180.000} C_DIS
LIN {X 54.089,Y 107.623,Z 72.500,A 180.000,B 0.000,C 180.000} C_DIS
LIN {X 54.171,Y 107.684,Z 72.500,A 180.000,B 0.000,C 180.000} C_DIS
LIN {X 54.344,Y 107.802,Z 72.500,A 180.000,B 0.000,C 180.000} C_DIS
LIN {X 54.707,Y 108.025,Z 72.500,A 180.000,B 0.000,C 180.000} C_DIS
LIN {X 54.886,Y 108.128,Z 72.500,A 180.000,B 0.000,C 180.000} C_DIS
LIN {X 54.947,Y 108.159,Z 72.500,A 180.000,B 0.000,C 180.000} C_DIS
LIN {X 55.304,Y 108.338,Z 72.500,A 180.000,B 0.000,C 180.000} C_DIS
LIN {X 55.422,Y 108.394,Z 72.500,A 180.000,B 0.000,C 180.000} C_DIS
LIN {X 55.601,Y 108.467,Z 72.500,A 180.000,B 0.000,C 180.000} C_DIS
LIN {X 55.779,Y 108.538,Z 72.500,A 180.000,B 0.000,C 180.000} C_DIS
LIN {X 55.958,Y 108.608,Z 72.500,A 180.000,B 0.000,C 180.000} C_DIS
LIN {X 56.137,Y 108.669,Z 72.500,A 180.000,B 0.000,C 180.000} C_DIS
LIN {X 56.225,Y 108.695,Z 72.500,A 180.000,B 0.000,C 180.000} C_DIS
LIN {X 56.495,Y 108.775,Z 72.500,A 180.000,B 0.000,C 180.000} C_DIS
LIN {X 56.673,Y 108.826,Z 72.500,A 180.000,B 0.000,C 180.000} C_DIS
LIN {X 56.852,Y 108.865,Z 72.500,A 180.000,B 0.000,C 180.000} C_DIS
LIN {X 57.210,Y 108.937,Z 72.500,A 180.000,B 0.000,C 180.000} C_DIS
LIN {X 57.388,Y 108.967,Z 72.500,A 180.000,B 0.000,C 180.000} C_DIS
LIN {X 57.567,Y 108.988,Z 72.500,A 180.000,B 0.000,C 180.000} C_DIS
LIN {X 57.746,Y 109.008,Z 72.500,A 180.000,B 0.000,C 180.000} C_DIS
LIN {X 57.925,Y 109.027,Z 72.500,A 180.000,B 0.000,C 180.000} C_DIS
LIN {X 58.103,Y 109.038,Z 72.500,A 180.000,B 0.000,C 180.000} C_DIS
LIN {X 58.461,Y 109.046,Z 72.500,A 180.000,B 0.000,C 180.000} C_DIS
LIN {X 58.640,Y 109.049,Z 72.500,A 180.000,B 0.000,C 180.000} C_DIS
LIN {X 58.819,Y 109.041,Z 72.500,A 180.000,B 0.000,C 180.000} C_DIS
LIN {X 59.176,Y 109.017,Z 72.500,A 180.000,B 0.000,C 180.000} C_DIS
LIN {X 59.355,Y 109.001,Z 72.500,A 180.000,B 0.000,C 180.000} C_DIS
LIN {X 59.534,Y 108.975,Z 72.500,A 180.000,B 0.000,C 180.000} C_DIS
LIN {X 59.891,Y 108.919,Z 72.500,A 180.000,B 0.000,C 180.000} C_DIS
LIN {X 60.070,Y 108.884,Z 72.500,A 180.000,B 0.000,C 180.000} C_DIS
LIN {X 60.111,Y 108.874,Z 72.500,A 180.000,B 0.000,C 180.000} C_DIS
LIN {X 60.427,Y 108.796,Z 72.500,A 180.000,B 0.000,C 180.000} C_DIS
LIN {X 60.606,Y 108.750,Z 72.500,A 180.000,B 0.000,C 180.000} C_DIS
LIN {X 60.778,Y 108.695,Z 72.500,A 180.000,B 0.000,C 180.000} C_DIS
LIN {X 61.143,Y 108.570,Z 72.500,A 180.000,B 0.000,C 180.000} C_DIS
LIN {X 61.287,Y 108.517,Z 72.500,A 180.000,B 0.000,C 180.000} C_DIS
LIN {X 61.321,Y 108.503,Z 72.500,A 180.000,B 0.000,C 180.000} C_DIS
LIN {X 61.500,Y 108.424,Z 72.500,A 180.000,B 0.000,C 180.000} C_DIS
LIN {X 61.692,Y 108.338,Z 72.500,A 180.000,B 0.000,C 180.000} C_DIS
LIN {X 61.858,Y 108.262,Z 72.500,A 180.000,B 0.000,C 180.000} C_DIS
LIN {X 62.036,Y 108.167,Z 72.500,A 180.000,B 0.000,C 180.000} C_DIS
LIN {X 62.371,Y 107.980,Z 72.500,A 180.000,B 0.000,C 180.000} C_DIS
LIN {X 62.394,Y 107.967,Z 72.500,A 180.000,B 0.000,C 180.000} C_DIS
LIN {X 62.573,Y 107.855,Z 72.500,A 180.000,B 0.000,C 180.000} C_DIS
LIN {X 62.930,Y 107.612,Z 72.500,A 180.000,B 0.000,C 180.000} C_DIS
LIN {X 63.020,Y 107.548,Z 72.500,A 180.000,B 0.000,C 180.000} C_DIS
LIN {X 63.109,Y 107.478,Z 72.500,A 180.000,B 0.000,C 180.000} C_DIS
LIN {X 63.369,Y 107.265,Z 72.500,A 180.000,B 0.000,C 180.000} C_DIS
LIN {X 63.467,Y 107.185,Z 72.500,A 180.000,B 0.000,C 180.000} C_DIS
LIN {X 63.578,Y 107.086,Z 72.500,A 180.000,B 0.000,C 180.000} C_DIS
LIN {X 63.645,Y 107.021,Z 72.500,A 180.000,B 0.000,C 180.000} C_DIS
LIN {X 63.824,Y 106.847,Z 72.500,A 180.000,B 0.000,C 180.000} C_DIS
LIN {X 63.944,Y 106.729,Z 72.500,A 180.000,B 0.000,C 180.000} C_DIS
LIN {X 64.003,Y 106.669,Z 72.500,A 180.000,B 0.000,C 180.000} C_DIS
LIN {X 64.109,Y 106.550,Z 72.500,A 180.000,B 0.000,C 180.000} C_DIS
LIN {X 64.360,Y 106.256,Z 72.500,A 180.000,B 0.000,C 180.000} C_DIS
LIN {X 64.414,Y 106.193,Z 72.500,A 180.000,B 0.000,C 180.000} C_DIS
LIN {X 64.539,Y 106.026,Z 72.500,A 180.000,B 0.000,C 180.000} C_DIS
LIN {X 64.718,Y 105.776,Z 72.500,A 180.000,B 0.000,C 180.000} C_DIS
LIN {X 64.802,Y 105.656,Z 72.500,A 180.000,B 0.000,C 180.000} C_DIS
LIN {X 64.897,Y 105.507,Z 72.500,A 180.000,B 0.000,C 180.000} C_DIS
LIN {X 65.075,Y 105.203,Z 72.500,A 180.000,B 0.000,C 180.000} C_DIS
LIN {X 65.124,Y 105.120,Z 72.500,A 180.000,B 0.000,C 180.000} C_DIS
LIN {X 65.219,Y 104.941,Z 72.500,A 180.000,B 0.000,C 180.000} C_DIS
LIN {X 65.254,Y 104.866,Z 72.500,A 180.000,B 0.000,C 180.000} C_DIS
LIN {X 65.388,Y 104.584,Z 72.500,A 180.000,B 0.000,C 180.000} C_DIS
LIN {X 65.433,Y 104.488,Z 72.500,A 180.000,B 0.000,C 180.000} C_DIS
LIN {X 65.469,Y 104.405,Z 72.500,A 180.000,B 0.000,C 180.000} C_DIS
LIN {X 65.536,Y 104.226,Z 72.500,A 180.000,B 0.000,C 180.000} C_DIS
LIN {X 65.612,Y 104.022,Z 72.500,A 180.000,B 0.000,C 180.000} C_DIS
LIN {X 65.668,Y 103.869,Z 72.500,A 180.000,B 0.000,C 180.000} C_DIS
LIN {X 65.724,Y 103.690,Z 72.500,A 180.000,B 0.000,C 180.000} C_DIS
LIN {X 65.821,Y 103.332,Z 72.500,A 180.000,B 0.000,C 180.000} C_DIS
LIN {X 65.867,Y 103.153,Z 72.500,A 180.000,B 0.000,C 180.000} C_DIS
LIN {X 65.901,Y 102.975,Z 72.500,A 180.000,B 0.000,C 180.000} C_DIS
LIN {X 65.965,Y 102.617,Z 72.500,A 180.000,B 0.000,C 180.000} C_DIS
LIN {X 65.969,Y 102.592,Z 72.500,A 180.000,B 0.000,C 180.000} C_DIS
LIN {X 65.991,Y 102.438,Z 72.500,A 180.000,B 0.000,C 180.000} C_DIS
LIN {X 66.007,Y 102.260,Z 72.500,A 180.000,B 0.000,C 180.000} C_DIS
LIN {X 66.023,Y 102.081,Z 72.500,A 180.000,B 0.000,C 180.000} C_DIS
LIN {X 66.039,Y 101.902,Z 72.500,A 180.000,B 0.000,C 180.000} C_DIS
LIN {X 66.045,Y 101.723,Z 72.500,A 180.000,B 0.000,C 180.000} C_DIS
LIN {X 66.045,Y 101.366,Z 72.500,A 180.000,B 0.000,C 180.000} C_DIS
LIN {X 66.043,Y 101.187,Z 72.500,A 180.000,B 0.000,C 180.000} C_DIS
LIN {X 66.031,Y 101.008,Z 72.500,A 180.000,B 0.000,C 180.000} C_DIS
LIN {X 65.999,Y 100.651,Z 72.500,A 180.000,B 0.000,C 180.000} C_DIS
LIN {X 65.980,Y 100.472,Z 72.500,A 180.000,B 0.000,C 180.000} C_DIS
LIN {X 65.969,Y 100.408,Z 72.500,A 180.000,B 0.000,C 180.000} C_DIS
LIN {X 65.949,Y 100.293,Z 72.500,A 180.000,B 0.000,C 180.000} C_DIS
LIN {X 65.917,Y 100.114,Z 72.500,A 180.000,B 0.000,C 180.000} C_DIS
LIN {X 65.885,Y 99.936,Z 72.500,A 180.000,B 0.000,C 180.000} C_DIS
LIN {X 65.845,Y 99.757,Z 72.500,A 180.000,B 0.000,C 180.000} C_DIS
LIN {X 65.796,Y 99.578,Z 72.500,A 180.000,B 0.000,C 180.000} C_DIS
LIN {X 65.748,Y 99.399,Z 72.500,A 180.000,B 0.000,C 180.000} C_DIS
LIN {X 65.698,Y 99.221,Z 72.500,A 180.000,B 0.000,C 180.000} C_DIS
LIN {X 65.635,Y 99.042,Z 72.500,A 180.000,B 0.000,C 180.000} C_DIS
LIN {X 65.503,Y 98.684,Z 72.500,A 180.000,B 0.000,C 180.000} C_DIS
LIN {X 65.433,Y 98.512,Z 72.500,A 180.000,B 0.000,C 180.000} C_DIS
LIN {X 65.430,Y 98.505,Z 72.500,A 180.000,B 0.000,C 180.000} C_DIS
LIN {X 65.346,Y 98.327,Z 72.500,A 180.000,B 0.000,C 180.000} C_DIS
LIN {X 65.254,Y 98.134,Z 72.500,A 180.000,B 0.000,C 180.000} C_DIS
LIN {X 65.174,Y 97.969,Z 72.500,A 180.000,B 0.000,C 180.000} C_DIS
LIN {X 65.075,Y 97.797,Z 72.500,A 180.000,B 0.000,C 180.000} C_DIS
LIN {X 64.897,Y 97.493,Z 72.500,A 180.000,B 0.000,C 180.000} C_DIS
LIN {X 64.861,Y 97.433,Z 72.500,A 180.000,B 0.000,C 180.000} C_DIS
LIN {X 64.739,Y 97.254,Z 72.500,A 180.000,B 0.000,C 180.000} C_DIS
LIN {X 64.539,Y 96.974,Z 72.500,A 180.000,B 0.000,C 180.000} C_DIS
LIN {X 64.484,Y 96.897,Z 72.500,A 180.000,B 0.000,C 180.000} C_DIS
LIN {X 64.360,Y 96.744,Z 72.500,A 180.000,B 0.000,C 180.000} C_DIS
LIN {X 64.182,Y 96.535,Z 72.500,A 180.000,B 0.000,C 180.000} C_DIS
LIN {X 64.030,Y 96.360,Z 72.500,A 180.000,B 0.000,C 180.000} C_DIS
LIN {X 64.003,Y 96.331,Z 72.500,A 180.000,B 0.000,C 180.000} C_DIS
LIN {X 63.853,Y 96.181,Z 72.500,A 180.000,B 0.000,C 180.000} C_DIS
LIN {X 63.645,Y 95.979,Z 72.500,A 180.000,B 0.000,C 180.000} C_DIS
LIN {X 63.477,Y 95.824,Z 72.500,A 180.000,B 0.000,C 180.000} C_DIS
LIN {X 63.467,Y 95.815,Z 72.500,A 180.000,B 0.000,C 180.000} C_DIS
LIN {X 63.288,Y 95.669,Z 72.500,A 180.000,B 0.000,C 180.000} C_DIS
LIN {X 63.109,Y 95.522,Z 72.500,A 180.000,B 0.000,C 180.000} C_DIS
LIN {X 63.038,Y 95.466,Z 72.500,A 180.000,B 0.000,C 180.000} C_DIS
LIN {X 62.930,Y 95.388,Z 72.500,A 180.000,B 0.000,C 180.000} C_DIS
LIN {X 62.573,Y 95.145,Z 72.500,A 180.000,B 0.000,C 180.000} C_DIS
LIN {X 62.518,Y 95.109,Z 72.500,A 180.000,B 0.000,C 180.000} C_DIS
LIN {X 62.394,Y 95.033,Z 72.500,A 180.000,B 0.000,C 180.000} C_DIS
LIN {X 62.210,Y 94.930,Z 72.500,A 180.000,B 0.000,C 180.000} C_DIS
LIN {X 62.036,Y 94.833,Z 72.500,A 180.000,B 0.000,C 180.000} C_DIS
LIN {X 61.885,Y 94.751,Z 72.500,A 180.000,B 0.000,C 180.000} C_DIS
LIN {X 61.858,Y 94.738,Z 72.500,A 180.000,B 0.000,C 180.000} C_DIS
LIN {X 61.679,Y 94.656,Z 72.500,A 180.000,B 0.000,C 180.000} C_DIS
LIN {X 61.491,Y 94.573,Z 72.500,A 180.000,B 0.000,C 180.000} C_DIS
LIN {X 61.321,Y 94.497,Z 72.500,A 180.000,B 0.000,C 180.000} C_DIS
LIN {X 61.143,Y 94.430,Z 72.500,A 180.000,B 0.000,C 180.000} C_DIS
LIN {X 60.785,Y 94.307,Z 72.500,A 180.000,B 0.000,C 180.000} C_DIS
LIN {X 60.606,Y 94.250,Z 72.500,A 180.000,B 0.000,C 180.000} C_DIS
LIN {X 60.470,Y 94.215,Z 72.500,A 180.000,B 0.000,C 180.000} C_DIS
LIN {X 60.249,Y 94.160,Z 72.500,A 180.000,B 0.000,C 180.000} C_DIS
LIN {X 60.070,Y 94.116,Z 72.500,A 180.000,B 0.000,C 180.000} C_DIS
LIN {X 59.891,Y 94.081,Z 72.500,A 180.000,B 0.000,C 180.000} C_DIS
LIN {X 59.534,Y 94.025,Z 72.500,A 180.000,B 0.000,C 180.000} C_DIS
LIN {X 59.355,Y 93.999,Z 72.500,A 180.000,B 0.000,C 180.000} C_DIS
LIN {X 59.176,Y 93.983,Z 72.500,A 180.000,B 0.000,C 180.000} C_DIS
LIN {X 58.819,Y 93.959,Z 72.500,A 180.000,B 0.000,C 180.000} C_DIS
LIN {X 58.640,Y 93.951,Z 72.500,A 180.000,B 0.000,C 180.000} C_DIS
LIN {X 58.461,Y 93.954,Z 72.500,A 180.000,B 0.000,C 180.000} C_DIS
LIN {X 58.103,Y 93.962,Z 72.500,A 180.000,B 0.000,C 180.000} C_DIS
LIN {X 57.925,Y 93.973,Z 72.500,A 180.000,B 0.000,C 180.000} C_DIS
LIN {X 57.746,Y 93.992,Z 72.500,A 180.000,B 0.000,C 180.000} C_DIS
LIN {X 57.567,Y 94.012,Z 72.500,A 180.000,B 0.000,C 180.000} C_DIS
LIN {X 57.388,Y 94.033,Z 72.500,A 180.000,B 0.000,C 180.000} C_DIS
LIN {X 57.363,Y 94.036,Z 72.500,A 180.000,B 0.000,C 180.000} C_DIS
LIN {X 57.210,Y 94.063,Z 72.500,A 180.000,B 0.000,C 180.000} C_DIS
LIN {X 56.852,Y 94.135,Z 72.500,A 180.000,B 0.000,C 180.000} C_DIS
LIN {X 56.673,Y 94.174,Z 72.500,A 180.000,B 0.000,C 180.000} C_DIS
LIN {X 56.528,Y 94.215,Z 72.500,A 180.000,B 0.000,C 180.000} C_DIS
LIN {X 56.316,Y 94.278,Z 72.500,A 180.000,B 0.000,C 180.000} C_DIS
LIN {X 56.137,Y 94.331,Z 72.500,A 180.000,B 0.000,C 180.000} C_DIS
LIN {X 55.958,Y 94.392,Z 72.500,A 180.000,B 0.000,C 180.000} C_DIS
LIN {X 55.953,Y 94.394,Z 72.500,A 180.000,B 0.000,C 180.000} C_DIS
LIN {X 55.779,Y 94.462,Z 72.500,A 180.000,B 0.000,C 180.000} C_DIS
LIN {X 55.601,Y 94.533,Z 72.500,A 180.000,B 0.000,C 180.000} C_DIS
LIN {X 55.501,Y 94.573,Z 72.500,A 180.000,B 0.000,C 180.000} C_DIS
LIN {X 55.422,Y 94.606,Z 72.500,A 180.000,B 0.000,C 180.000} C_DIS
LIN {X 55.243,Y 94.693,Z 72.500,A 180.000,B 0.000,C 180.000} C_DIS
LIN {X 55.064,Y 94.782,Z 72.500,A 180.000,B 0.000,C 180.000} C_DIS
LIN {X 54.886,Y 94.872,Z 72.500,A 180.000,B 0.000,C 180.000} C_DIS
LIN {X 54.781,Y 94.930,Z 72.500,A 180.000,B 0.000,C 180.000} C_DIS
LIN {X 54.707,Y 94.975,Z 72.500,A 180.000,B 0.000,C 180.000} C_DIS
LIN {X 54.349,Y 95.195,Z 72.500,A 180.000,B 0.000,C 180.000} C_DIS
LIN {X 54.210,Y 95.288,Z 72.500,A 180.000,B 0.000,C 180.000} C_DIS
LIN {X 54.171,Y 95.316,Z 72.500,A 180.000,B 0.000,C 180.000} C_DIS
LIN {X 53.970,Y 95.466,Z 72.500,A 180.000,B 0.000,C 180.000} C_DIS
LIN {X 53.813,Y 95.583,Z 72.500,A 180.000,B 0.000,C 180.000} C_DIS
LIN {X 53.733,Y 95.645,Z 72.500,A 180.000,B 0.000,C 180.000} C_DIS
LIN {X 53.634,Y 95.729,Z 72.500,A 180.000,B 0.000,C 180.000} C_DIS
LIN {X 53.329,Y 96.003,Z 72.500,A 180.000,B 0.000,C 180.000} C_DIS
LIN {X 53.277,Y 96.050,Z 72.500,A 180.000,B 0.000,C 180.000} C_DIS
LIN {X 53.144,Y 96.181,Z 72.500,A 180.000,B 0.000,C 180.000} C_DIS
LIN {X 52.919,Y 96.421,Z 72.500,A 180.000,B 0.000,C 180.000} C_DIS
LIN {X 52.810,Y 96.539,Z 72.500,A 180.000,B 0.000,C 180.000} C_DIS
LIN {X 52.740,Y 96.619,Z 72.500,A 180.000,B 0.000,C 180.000} C_DIS
LIN {X 52.662,Y 96.718,Z 72.500,A 180.000,B 0.000,C 180.000} C_DIS
LIN {X 52.522,Y 96.897,Z 72.500,A 180.000,B 0.000,C 180.000} C_DIS
LIN {X 52.383,Y 97.075,Z 72.500,A 180.000,B 0.000,C 180.000} C_DIS
LIN {X 52.261,Y 97.254,Z 72.500,A 180.000,B 0.000,C 180.000} C_DIS
LIN {X 52.145,Y 97.433,Z 72.500,A 180.000,B 0.000,C 180.000} C_DIS
LIN {X 52.029,Y 97.612,Z 72.500,A 180.000,B 0.000,C 180.000} C_DIS
LIN {X 52.025,Y 97.618,Z 72.500,A 180.000,B 0.000,C 180.000} C_DIS
LIN {X 51.927,Y 97.790,Z 72.500,A 180.000,B 0.000,C 180.000} C_DIS
LIN {X 51.737,Y 98.148,Z 72.500,A 180.000,B 0.000,C 180.000} C_DIS
LIN {X 51.668,Y 98.287,Z 72.500,A 180.000,B 0.000,C 180.000} C_DIS
LIN {X 51.650,Y 98.327,Z 72.500,A 180.000,B 0.000,C 180.000} C_DIS
LIN {X 51.574,Y 98.505,Z 72.500,A 180.000,B 0.000,C 180.000} C_DIS
LIN {X 51.489,Y 98.708,Z 72.500,A 180.000,B 0.000,C 180.000} C_DIS
LIN {X 51.426,Y 98.863,Z 72.500,A 180.000,B 0.000,C 180.000} C_DIS
LIN {X 51.365,Y 99.042,Z 72.500,A 180.000,B 0.000,C 180.000} C_DIS
LIN {X 51.250,Y 99.399,Z 72.500,A 180.000,B 0.000,C 180.000} C_DIS
LIN {X 51.199,Y 99.578,Z 72.500,A 180.000,B 0.000,C 180.000} C_DIS
LIN {X 51.159,Y 99.757,Z 72.500,A 180.000,B 0.000,C 180.000} C_DIS
LIN {X 51.118,Y 99.936,Z 72.500,A 180.000,B 0.000,C 180.000} C_DIS
LIN {X 51.079,Y 100.114,Z 72.500,A 180.000,B 0.000,C 180.000} C_DIS
LIN {X 51.049,Y 100.293,Z 72.500,A 180.000,B 0.000,C 180.000} C_DIS
LIN {X 51.001,Y 100.651,Z 72.500,A 180.000,B 0.000,C 180.000} C_DIS
LIN {X 50.980,Y 100.829,Z 72.500,A 180.000,B 0.000,C 180.000} C_DIS
LIN {X 50.969,Y 101.008,Z 72.500,A 180.000,B 0.000,C 180.000} C_DIS
LIN {X 50.953,Y 101.385,Z 72.500,A 180.000,B 0.000,C 180.000} C_DIS
LIN {X 50.950,Y 101.545,Z 72.500,A 180.000,B 0.000,C 180.000} C_DIS
LIN {X 50.953,Y 101.615,Z 72.500,A 180.000,B 0.000,C 180.000} C_DIS
LIN {X 50.965,Y 101.902,Z 72.500,A 180.000,B 0.000,C 180.000} C_DIS
LIN {X 50.973,Y 102.081,Z 72.500,A 180.000,B 0.000,C 180.000} C_DIS
LIN {X 50.989,Y 102.260,Z 72.500,A 180.000,B 0.000,C 180.000} C_DIS
LIN {X 51.013,Y 102.438,Z 72.500,A 180.000,B 0.000,C 180.000} C_DIS
LIN {X 51.037,Y 102.617,Z 72.500,A 180.000,B 0.000,C 180.000} C_DIS
LIN {X 51.062,Y 102.796,Z 72.500,A 180.000,B 0.000,C 180.000} C_DIS
LIN {X 51.098,Y 102.975,Z 72.500,A 180.000,B 0.000,C 180.000} C_DIS
LIN {X 51.179,Y 103.332,Z 72.500,A 180.000,B 0.000,C 180.000} C_DIS
LIN {X 51.223,Y 103.511,Z 72.500,A 180.000,B 0.000,C 180.000} C_DIS
LIN {X 51.279,Y 103.690,Z 72.500,A 180.000,B 0.000,C 180.000} C_DIS
LIN {X 51.336,Y 103.869,Z 72.500,A 180.000,B 0.000,C 180.000} C_DIS
LIN {X 51.393,Y 104.047,Z 72.500,A 180.000,B 0.000,C 180.000} C_DIS
LIN {X 51.461,Y 104.226,Z 72.500,A 180.000,B 0.000,C 180.000} C_DIS
LIN {X 51.612,Y 104.584,Z 72.500,A 180.000,B 0.000,C 180.000} C_DIS
LIN {X 51.668,Y 104.713,Z 72.500,A 180.000,B 0.000,C 180.000} C_DIS
LIN {X 51.691,Y 104.762,Z 72.500,A 180.000,B 0.000,C 180.000} C_DIS
LIN {X 51.785,Y 104.941,Z 72.500,A 180.000,B 0.000,C 180.000} C_DIS
LIN {X 51.879,Y 105.120,Z 72.500,A 180.000,B 0.000,C 180.000} C_DIS
LIN {X 51.975,Y 105.299,Z 72.500,A 180.000,B 0.000,C 180.000} C_DIS
LIN {X 51.998,Y 105.336,Z 72.500,A 180.000,B 0.000,C 180.000} C_DIS
; Link Move Starts
LIN {X 52.167,Y 105.602,Z 72.500,A 180.000,B 0.000,C 180.000} C_DIS
LIN {X 52.340,Y 105.865,Z 72.499,A 180.000,B 0.000,C 180.000} C_DIS
LIN {X 52.531,Y 106.115,Z 72.498,A 180.000,B 0.000,C 180.000} C_DIS
LIN {X 52.726,Y 106.363,Z 72.496,A 180.000,B 0.000,C 180.000} C_DIS
LIN {X 52.936,Y 106.597,Z 72.494,A 180.000,B 0.000,C 180.000} C_DIS
LIN {X 53.152,Y 106.827,Z 72.491,A 180.000,B 0.000,C 180.000} C_DIS
LIN {X 53.380,Y 107.044,Z 72.488,A 180.000,B 0.000,C 180.000} C_DIS
LIN {X 53.615,Y 107.254,Z 72.485,A 180.000,B 0.000,C 180.000} C_DIS
LIN {X 53.735,Y 107.356,Z 72.483,A 180.000,B 0.000,C 180.000} C_DIS
LIN {X 53.860,Y 107.452,Z 72.481,A 180.000,B 0.000,C 180.000} C_DIS
LIN {X 54.112,Y 107.640,Z 72.477,A 180.000,B 0.000,C 180.000} C_DIS
LIN {X 54.240,Y 107.733,Z 72.474,A 180.000,B 0.000,C 180.000} C_DIS
LIN {X 54.372,Y 107.819,Z 72.472,A 180.000,B 0.000,C 180.000} C_DIS
LIN {X 54.506,Y 107.901,Z 72.469,A 180.000,B 0.000,C 180.000} C_DIS
LIN {X 54.640,Y 107.984,Z 72.467,A 180.000,B 0.000,C 180.000} C_DIS
LIN {X 54.774,Y 108.066,Z 72.464,A 180.000,B 0.000,C 180.000} C_DIS
LIN {X 54.913,Y 108.142,Z 72.461,A 180.000,B 0.000,C 180.000} C_DIS
LIN {X 55.053,Y 108.212,Z 72.459,A 180.000,B 0.000,C 180.000} C_DIS
LIN {X 55.194,Y 108.283,Z 72.456,A 180.000,B 0.000,C 180.000} C_DIS
LIN {X 55.335,Y 108.353,Z 72.452,A 180.000,B 0.000,C 180.000} C_DIS
LIN {X 55.478,Y 108.418,Z 72.449,A 180.000,B 0.000,C 180.000} C_DIS
LIN {X 55.625,Y 108.477,Z 72.446,A 180.000,B 0.000,C 180.000} C_DIS
LIN {X 55.771,Y 108.534,Z 72.443,A 180.000,B 0.000,C 180.000} C_DIS
LIN {X 55.918,Y 108.592,Z 72.439,A 180.000,B 0.000,C 180.000} C_DIS
LIN {X 56.066,Y 108.647,Z 72.436,A 180.000,B 0.000,C 180.000} C_DIS
LIN {X 56.216,Y 108.693,Z 72.432,A 180.000,B 0.000,C 180.000} C_DIS
LIN {X 56.367,Y 108.737,Z 72.428,A 180.000,B 0.000,C 180.000} C_DIS
LIN {X 56.518,Y 108.782,Z 72.425,A 180.000,B 0.000,C 180.000} C_DIS
LIN {X 56.670,Y 108.825,Z 72.421,A 180.000,B 0.000,C 180.000} C_DIS
LIN {X 56.824,Y 108.859,Z 72.417,A 180.000,B 0.000,C 180.000} C_DIS
LIN {X 56.978,Y 108.890,Z 72.413,A 180.000,B 0.000,C 180.000} C_DIS
LIN {X 57.132,Y 108.921,Z 72.409,A 180.000,B 0.000,C 180.000} C_DIS
LIN {X 57.287,Y 108.952,Z 72.405,A 180.000,B 0.000,C 180.000} C_DIS
LIN {X 57.443,Y 108.974,Z 72.400,A 180.000,B 0.000,C 180.000} C_DIS
LIN {X 57.599,Y 108.991,Z 72.396,A 180.000,B 0.000,C 180.000} C_DIS
LIN {X 57.756,Y 109.009,Z 72.392,A 180.000,B 0.000,C 180.000} C_DIS
LIN {X 57.912,Y 109.026,Z 72.387,A 180.000,B 0.000,C 180.000} C_DIS
LIN {X 58.070,Y 109.037,Z 72.383,A 180.000,B 0.000,C 180.000} C_DIS
LIN {X 58.227,Y 109.041,Z 72.378,A 180.000,B 0.000,C 180.000} C_DIS
LIN {X 58.384,Y 109.044,Z 72.373,A 180.000,B 0.000,C 180.000} C_DIS
LIN {X 58.542,Y 109.048,Z 72.369,A 180.000,B 0.000,C 180.000} C_DIS
LIN {X 58.699,Y 109.047,Z 72.364,A 180.000,B 0.000,C 180.000} C_DIS
LIN {X 58.857,Y 109.038,Z 72.359,A 180.000,B 0.000,C 180.000} C_DIS
LIN {X 59.014,Y 109.028,Z 72.354,A 180.000,B 0.000,C 180.000} C_DIS
LIN {X 59.092,Y 109.022,Z 72.351,A 180.000,B 0.000,C 180.000} C_DIS
LIN {X 59.171,Y 109.017,Z 72.349,A 180.000,B 0.000,C 180.000} C_DIS
LIN {X 59.250,Y 109.012,Z 72.346,A 180.000,B 0.000,C 180.000} C_DIS
LIN {X 59.328,Y 109.004,Z 72.344,A 180.000,B 0.000,C 180.000} C_DIS
LIN {X 59.406,Y 108.995,Z 72.341,A 180.000,B 0.000,C 180.000} C_DIS
LIN {X 59.484,Y 108.983,Z 72.339,A 180.000,B 0.000,C 180.000} C_DIS
LIN {X 59.562,Y 108.971,Z 72.336,A 180.000,B 0.000,C 180.000} C_DIS
LIN {X 59.717,Y 108.946,Z 72.331,A 180.000,B 0.000,C 180.000} C_DIS
LIN {X 59.873,Y 108.922,Z 72.325,A 180.000,B 0.000,C 180.000} C_DIS
LIN {X 59.951,Y 108.909,Z 72.323,A 180.000,B 0.000,C 180.000} C_DIS
LIN {X 60.028,Y 108.894,Z 72.320,A 180.000,B 0.000,C 180.000} C_DIS
LIN {X 60.105,Y 108.876,Z 72.317,A 180.000,B 0.000,C 180.000} C_DIS
LIN {X 60.257,Y 108.838,Z 72.312,A 180.000,B 0.000,C 180.000} C_DIS
LIN {X 60.487,Y 108.781,Z 72.304,A 180.000,B 0.000,C 180.000} C_DIS
LIN {X 60.563,Y 108.762,Z 72.301,A 180.000,B 0.000,C 180.000} C_DIS
LIN {X 60.639,Y 108.741,Z 72.298,A 180.000,B 0.000,C 180.000} C_DIS
LIN {X 60.714,Y 108.717,Z 72.296,A 180.000,B 0.000,C 180.000} C_DIS
LIN {X 60.789,Y 108.692,Z 72.293,A 180.000,B 0.000,C 180.000} C_DIS
LIN {X 60.938,Y 108.640,Z 72.287,A 180.000,B 0.000,C 180.000} C_DIS
LIN {X 61.012,Y 108.615,Z 72.285,A 180.000,B 0.000,C 180.000} C_DIS
LIN {X 61.161,Y 108.563,Z 72.279,A 180.000,B 0.000,C 180.000} C_DIS
LIN {X 61.235,Y 108.537,Z 72.276,A 180.000,B 0.000,C 180.000} C_DIS
LIN {X 61.308,Y 108.508,Z 72.274,A 180.000,B 0.000,C 180.000} C_DIS
LIN {X 61.381,Y 108.477,Z 72.271,A 180.000,B 0.000,C 180.000} C_DIS
LIN {X 61.525,Y 108.413,Z 72.265,A 180.000,B 0.000,C 180.000} C_DIS
LIN {X 61.596,Y 108.380,Z 72.263,A 180.000,B 0.000,C 180.000} C_DIS
LIN {X 61.740,Y 108.316,Z 72.257,A 180.000,B 0.000,C 180.000} C_DIS
LIN {X 61.812,Y 108.284,Z 72.254,A 180.000,B 0.000,C 180.000} C_DIS
LIN {X 61.883,Y 108.250,Z 72.252,A 180.000,B 0.000,C 180.000} C_DIS
LIN {X 61.953,Y 108.213,Z 72.249,A 180.000,B 0.000,C 180.000} C_DIS
LIN {X 62.022,Y 108.175,Z 72.246,A 180.000,B 0.000,C 180.000} C_DIS
LIN {X 62.228,Y 108.060,Z 72.238,A 180.000,B 0.000,C 180.000} C_DIS
LIN {X 62.366,Y 107.983,Z 72.232,A 180.000,B 0.000,C 180.000} C_DIS
LIN {X 62.434,Y 107.944,Z 72.230,A 180.000,B 0.000,C 180.000} C_DIS
LIN {X 62.501,Y 107.903,Z 72.227,A 180.000,B 0.000,C 180.000} C_DIS
LIN {X 62.567,Y 107.859,Z 72.224,A 180.000,B 0.000,C 180.000} C_DIS
LIN {X 62.892,Y 107.638,Z 72.210,A 180.000,B 0.000,C 180.000} C_DIS
LIN {X 62.957,Y 107.593,Z 72.208,A 180.000,B 0.000,C 180.000} C_DIS
LIN {X 63.021,Y 107.547,Z 72.205,A 180.000,B 0.000,C 180.000} C_DIS
LIN {X 63.083,Y 107.499,Z 72.202,A 180.000,B 0.000,C 180.000} C_DIS
LIN {X 63.144,Y 107.449,Z 72.199,A 180.000,B 0.000,C 180.000} C_DIS
LIN {X 63.205,Y 107.399,Z 72.197,A 180.000,B 0.000,C 180.000} C_DIS
LIN {X 63.327,Y 107.299,Z 72.191,A 180.000,B 0.000,C 180.000} C_DIS
LIN {X 63.449,Y 107.200,Z 72.186,A 180.000,B 0.000,C 180.000} C_DIS
LIN {X 63.509,Y 107.149,Z 72.183,A 180.000,B 0.000,C 180.000} C_DIS
LIN {X 63.568,Y 107.096,Z 72.180,A 180.000,B 0.000,C 180.000} C_DIS
LIN {X 63.625,Y 107.042,Z 72.177,A 180.000,B 0.000,C 180.000} C_DIS
LIN {X 63.681,Y 106.987,Z 72.175,A 180.000,B 0.000,C 180.000} C_DIS
LIN {X 63.794,Y 106.877,Z 72.169,A 180.000,B 0.000,C 180.000} C_DIS
LIN {X 63.906,Y 106.766,Z 72.164,A 180.000,B 0.000,C 180.000} C_DIS
LIN {X 63.962,Y 106.711,Z 72.161,A 180.000,B 0.000,C 180.000} C_DIS
LIN {X 64.017,Y 106.654,Z 72.158,A 180.000,B 0.000,C 180.000} C_DIS
LIN {X 64.070,Y 106.596,Z 72.155,A 180.000,B 0.000,C 180.000} C_DIS
LIN {X 64.121,Y 106.536,Z 72.153,A 180.000,B 0.000,C 180.000} C_DIS
LIN {X 64.274,Y 106.357,Z 72.144,A 180.000,B 0.000,C 180.000} C_DIS
LIN {X 64.377,Y 106.237,Z 72.139,A 180.000,B 0.000,C 180.000} C_DIS
LIN {X 64.427,Y 106.176,Z 72.136,A 180.000,B 0.000,C 180.000} C_DIS
LIN {X 64.476,Y 106.114,Z 72.133,A 180.000,B 0.000,C 180.000} C_DIS
LIN {X 64.522,Y 106.051,Z 72.131,A 180.000,B 0.000,C 180.000} C_DIS
LIN {X 64.659,Y 105.858,Z 72.122,A 180.000,B 0.000,C 180.000} C_DIS
LIN {X 64.751,Y 105.730,Z 72.117,A 180.000,B 0.000,C 180.000} C_DIS
LIN {X 64.796,Y 105.666,Z 72.114,A 180.000,B 0.000,C 180.000} C_DIS
LIN {X 64.840,Y 105.600,Z 72.111,A 180.000,B 0.000,C 180.000} C_DIS
LIN {X 64.881,Y 105.533,Z 72.109,A 180.000,B 0.000,C 180.000} C_DIS
LIN {X 64.921,Y 105.465,Z 72.106,A 180.000,B 0.000,C 180.000} C_DIS
LIN {X 65.121,Y 105.126,Z 72.092,A 180.000,B 0.000,C 180.000} C_DIS
LIN {X 65.159,Y 105.057,Z 72.089,A 180.000,B 0.000,C 180.000} C_DIS
LIN {X 65.196,Y 104.988,Z 72.087,A 180.000,B 0.000,C 180.000} C_DIS
LIN {X 65.230,Y 104.917,Z 72.084,A 180.000,B 0.000,C 180.000} C_DIS
LIN {X 65.399,Y 104.561,Z 72.070,A 180.000,B 0.000,C 180.000} C_DIS
LIN {X 65.432,Y 104.489,Z 72.067,A 180.000,B 0.000,C 180.000} C_DIS
LIN {X 65.464,Y 104.417,Z 72.065,A 180.000,B 0.000,C 180.000} C_DIS
LIN {X 65.493,Y 104.344,Z 72.062,A 180.000,B 0.000,C 180.000} C_DIS
LIN {X 65.520,Y 104.270,Z 72.059,A 180.000,B 0.000,C 180.000} C_DIS
LIN {X 65.657,Y 103.901,Z 72.045,A 180.000,B 0.000,C 180.000} C_DIS
LIN {X 65.683,Y 103.827,Z 72.043,A 180.000,B 0.000,C 180.000} C_DIS
LIN {X 65.706,Y 103.751,Z 72.040,A 180.000,B 0.000,C 180.000} C_DIS
LIN {X 65.727,Y 103.676,Z 72.037,A 180.000,B 0.000,C 180.000} C_DIS
LIN {X 65.831,Y 103.296,Z 72.023,A 180.000,B 0.000,C 180.000} C_DIS
LIN {X 65.851,Y 103.220,Z 72.021,A 180.000,B 0.000,C 180.000} C_DIS
LIN {X 65.869,Y 103.143,Z 72.018,A 180.000,B 0.000,C 180.000} C_DIS
LIN {X 65.885,Y 103.066,Z 72.015,A 180.000,B 0.000,C 180.000} C_DIS
LIN {X 65.899,Y 102.988,Z 72.012,A 180.000,B 0.000,C 180.000} C_DIS
LIN {X 65.968,Y 102.601,Z 71.999,A 180.000,B 0.000,C 180.000} C_DIS
LIN {X 65.980,Y 102.523,Z 71.996,A 180.000,B 0.000,C 180.000} C_DIS
LIN {X 65.990,Y 102.445,Z 71.993,A 180.000,B 0.000,C 180.000} C_DIS
LIN {X 65.998,Y 102.366,Z 71.990,A 180.000,B 0.000,C 180.000} C_DIS
LIN {X 66.033,Y 101.974,Z 71.977,A 180.000,B 0.000,C 180.000} C_DIS
LIN {X 66.039,Y 101.896,Z 71.974,A 180.000,B 0.000,C 180.000} C_DIS
LIN {X 66.043,Y 101.817,Z 71.971,A 180.000,B 0.000,C 180.000} C_DIS
LIN {X 66.045,Y 101.738,Z 71.968,A 180.000,B 0.000,C 180.000} C_DIS
LIN {X 66.045,Y 101.659,Z 71.966,A 180.000,B 0.000,C 180.000} C_DIS
LIN {X 66.045,Y 101.344,Z 71.955,A 180.000,B 0.000,C 180.000} C_DIS
LIN {X 66.045,Y 101.266,Z 71.952,A 180.000,B 0.000,C 180.000} C_DIS
LIN {X 66.043,Y 101.187,Z 71.949,A 180.000,B 0.000,C 180.000} C_DIS
LIN {X 66.039,Y 101.108,Z 71.946,A 180.000,B 0.000,C 180.000} C_DIS
LIN {X 66.033,Y 101.030,Z 71.944,A 180.000,B 0.000,C 180.000} C_DIS
LIN {X 65.998,Y 100.638,Z 71.930,A 180.000,B 0.000,C 180.000} C_DIS
LIN {X 65.991,Y 100.559,Z 71.927,A 180.000,B 0.000,C 180.000} C_DIS
LIN {X 65.981,Y 100.481,Z 71.924,A 180.000,B 0.000,C 180.000} C_DIS
LIN {X 65.969,Y 100.403,Z 71.922,A 180.000,B 0.000,C 180.000} C_DIS
LIN {X 65.955,Y 100.326,Z 71.919,A 180.000,B 0.000,C 180.000} C_DIS
LIN {X 65.899,Y 100.016,Z 71.908,A 180.000,B 0.000,C 180.000} C_DIS
LIN {X 65.885,Y 99.938,Z 71.905,A 180.000,B 0.000,C 180.000} C_DIS
LIN {X 65.870,Y 99.861,Z 71.902,A 180.000,B 0.000,C 180.000} C_DIS
LIN {X 65.852,Y 99.784,Z 71.900,A 180.000,B 0.000,C 180.000} C_DIS
LIN {X 65.832,Y 99.708,Z 71.897,A 180.000,B 0.000,C 180.000} C_DIS
LIN {X 65.728,Y 99.328,Z 71.883,A 180.000,B 0.000,C 180.000} C_DIS
LIN {X 65.707,Y 99.252,Z 71.880,A 180.000,B 0.000,C 180.000} C_DIS
LIN {X 65.684,Y 99.177,Z 71.878,A 180.000,B 0.000,C 180.000} C_DIS
LIN {X 65.658,Y 99.103,Z 71.875,A 180.000,B 0.000,C 180.000} C_DIS
LIN {X 65.631,Y 99.029,Z 71.872,A 180.000,B 0.000,C 180.000} C_DIS
LIN {X 65.521,Y 98.733,Z 71.861,A 180.000,B 0.000,C 180.000} C_DIS
LIN {X 65.494,Y 98.659,Z 71.858,A 180.000,B 0.000,C 180.000} C_DIS
LIN {X 65.465,Y 98.586,Z 71.856,A 180.000,B 0.000,C 180.000} C_DIS
LIN {X 65.434,Y 98.514,Z 71.853,A 180.000,B 0.000,C 180.000} C_DIS
LIN {X 65.400,Y 98.443,Z 71.850,A 180.000,B 0.000,C 180.000} C_DIS
LIN {X 65.232,Y 98.087,Z 71.836,A 180.000,B 0.000,C 180.000} C_DIS
LIN {X 65.198,Y 98.016,Z 71.834,A 180.000,B 0.000,C 180.000} C_DIS
LIN {X 65.161,Y 97.946,Z 71.831,A 180.000,B 0.000,C 180.000} C_DIS
LIN {X 65.122,Y 97.877,Z 71.828,A 180.000,B 0.000,C 180.000} C_DIS
LIN {X 65.043,Y 97.742,Z 71.823,A 180.000,B 0.000,C 180.000} C_DIS
LIN {X 64.963,Y 97.606,Z 71.817,A 180.000,B 0.000,C 180.000} C_DIS
LIN {X 64.923,Y 97.538,Z 71.814,A 180.000,B 0.000,C 180.000} C_DIS
LIN {X 64.883,Y 97.470,Z 71.812,A 180.000,B 0.000,C 180.000} C_DIS
LIN {X 64.842,Y 97.403,Z 71.809,A 180.000,B 0.000,C 180.000} C_DIS
LIN {X 64.798,Y 97.337,Z 71.806,A 180.000,B 0.000,C 180.000} C_DIS
LIN {X 64.753,Y 97.273,Z 71.803,A 180.000,B 0.000,C 180.000} C_DIS
LIN {X 64.707,Y 97.209,Z 71.801,A 180.000,B 0.000,C 180.000} C_DIS
LIN {X 64.616,Y 97.081,Z 71.795,A 180.000,B 0.000,C 180.000} C_DIS
LIN {X 64.524,Y 96.952,Z 71.790,A 180.000,B 0.000,C 180.000} C_DIS
LIN {X 64.478,Y 96.889,Z 71.787,A 180.000,B 0.000,C 180.000} C_DIS
LIN {X 64.430,Y 96.827,Z 71.784,A 180.000,B 0.000,C 180.000} C_DIS
LIN {X 64.379,Y 96.766,Z 71.781,A 180.000,B 0.000,C 180.000} C_DIS
LIN {X 64.328,Y 96.706,Z 71.779,A 180.000,B 0.000,C 180.000} C_DIS
LIN {X 64.226,Y 96.586,Z 71.773,A 180.000,B 0.000,C 180.000} C_DIS
LIN {X 64.123,Y 96.467,Z 71.768,A 180.000,B 0.000,C 180.000} C_DIS
LIN {X 64.072,Y 96.407,Z 71.765,A 180.000,B 0.000,C 180.000} C_DIS
LIN {X 64.019,Y 96.348,Z 71.762,A 180.000,B 0.000,C 180.000} C_DIS
LIN {X 63.965,Y 96.292,Z 71.759,A 180.000,B 0.000,C 180.000} C_DIS
LIN {X 63.909,Y 96.236,Z 71.757,A 180.000,B 0.000,C 180.000} C_DIS
LIN {X 63.796,Y 96.126,Z 71.751,A 180.000,B 0.000,C 180.000} C_DIS
LIN {X 63.627,Y 95.961,Z 71.743,A 180.000,B 0.000,C 180.000} C_DIS
LIN {X 63.570,Y 95.906,Z 71.740,A 180.000,B 0.000,C 180.000} C_DIS
LIN {X 63.512,Y 95.854,Z 71.737,A 180.000,B 0.000,C 180.000} C_DIS
LIN {X 63.452,Y 95.803,Z 71.735,A 180.000,B 0.000,C 180.000} C_DIS
LIN {X 63.330,Y 95.703,Z 71.729,A 180.000,B 0.000,C 180.000} C_DIS
LIN {X 63.147,Y 95.553,Z 71.721,A 180.000,B 0.000,C 180.000} C_DIS
LIN {X 63.086,Y 95.504,Z 71.718,A 180.000,B 0.000,C 180.000} C_DIS
LIN {X 63.024,Y 95.455,Z 71.715,A 180.000,B 0.000,C 180.000} C_DIS
LIN {X 62.960,Y 95.409,Z 71.713,A 180.000,B 0.000,C 180.000} C_DIS
LIN {X 62.895,Y 95.365,Z 71.710,A 180.000,B 0.000,C 180.000} C_DIS
LIN {X 62.765,Y 95.276,Z 71.704,A 180.000,B 0.000,C 180.000} C_DIS
LIN {X 62.700,Y 95.232,Z 71.702,A 180.000,B 0.000,C 180.000} C_DIS
LIN {X 62.570,Y 95.143,Z 71.696,A 180.000,B 0.000,C 180.000} C_DIS
LIN {X 62.504,Y 95.100,Z 71.693,A 180.000,B 0.000,C 180.000} C_DIS
LIN {X 62.437,Y 95.058,Z 71.691,A 180.000,B 0.000,C 180.000} C_DIS
LIN {X 62.369,Y 95.019,Z 71.688,A 180.000,B 0.000,C 180.000} C_DIS
LIN {X 62.231,Y 94.942,Z 71.682,A 180.000,B 0.000,C 180.000} C_DIS
LIN {X 62.094,Y 94.865,Z 71.677,A 180.000,B 0.000,C 180.000} C_DIS
LIN {X 62.025,Y 94.827,Z 71.674,A 180.000,B 0.000,C 180.000} C_DIS
LIN {X 61.956,Y 94.789,Z 71.672,A 180.000,B 0.000,C 180.000} C_DIS
LIN {X 61.886,Y 94.752,Z 71.669,A 180.000,B 0.000,C 180.000} C_DIS
LIN {X 61.815,Y 94.718,Z 71.666,A 180.000,B 0.000,C 180.000} C_DIS
LIN {X 61.744,Y 94.685,Z 71.664,A 180.000,B 0.000,C 180.000} C_DIS
LIN {X 61.672,Y 94.653,Z 71.661,A 180.000,B 0.000,C 180.000} C_DIS
LIN {X 61.600,Y 94.621,Z 71.659,A 180.000,B 0.000,C 180.000} C_DIS
LIN {X 61.528,Y 94.589,Z 71.656,A 180.000,B 0.000,C 180.000} C_DIS
LIN {X 61.456,Y 94.557,Z 71.654,A 180.000,B 0.000,C 180.000} C_DIS
LIN {X 61.384,Y 94.525,Z 71.651,A 180.000,B 0.000,C 180.000} C_DIS
LIN {X 61.312,Y 94.493,Z 71.649,A 180.000,B 0.000,C 180.000} C_DIS
LIN {X 61.165,Y 94.438,Z 71.644,A 180.000,B 0.000,C 180.000} C_DIS
LIN {X 61.016,Y 94.386,Z 71.639,A 180.000,B 0.000,C 180.000} C_DIS
LIN {X 60.867,Y 94.335,Z 71.634,A 180.000,B 0.000,C 180.000} C_DIS
LIN {X 60.718,Y 94.284,Z 71.629,A 180.000,B 0.000,C 180.000} C_DIS
LIN {X 60.567,Y 94.239,Z 71.624,A 180.000,B 0.000,C 180.000} C_DIS
LIN {X 60.414,Y 94.201,Z 71.620,A 180.000,B 0.000,C 180.000} C_DIS
LIN {X 60.261,Y 94.163,Z 71.615,A 180.000,B 0.000,C 180.000} C_DIS
LIN {X 60.108,Y 94.125,Z 71.611,A 180.000,B 0.000,C 180.000} C_DIS
LIN {X 59.954,Y 94.092,Z 71.606,A 180.000,B 0.000,C 180.000} C_DIS
LIN {X 59.799,Y 94.066,Z 71.602,A 180.000,B 0.000,C 180.000} C_DIS
LIN {X 59.643,Y 94.042,Z 71.597,A 180.000,B 0.000,C 180.000} C_DIS
LIN {X 59.488,Y 94.018,Z 71.593,A 180.000,B 0.000,C 180.000} C_DIS
LIN {X 59.332,Y 93.996,Z 71.589,A 180.000,B 0.000,C 180.000} C_DIS
LIN {X 59.175,Y 93.983,Z 71.585,A 180.000,B 0.000,C 180.000} C_DIS
LIN {X 59.018,Y 93.973,Z 71.581,A 180.000,B 0.000,C 180.000} C_DIS
LIN {X 58.860,Y 93.962,Z 71.577,A 180.000,B 0.000,C 180.000} C_DIS
LIN {X 58.703,Y 93.953,Z 71.573,A 180.000,B 0.000,C 180.000} C_DIS
LIN {X 58.546,Y 93.952,Z 71.570,A 180.000,B 0.000,C 180.000} C_DIS
LIN {X 58.388,Y 93.956,Z 71.566,A 180.000,B 0.000,C 180.000} C_DIS
LIN {X 58.231,Y 93.959,Z 71.562,A 180.000,B 0.000,C 180.000} C_DIS
LIN {X 58.073,Y 93.963,Z 71.559,A 180.000,B 0.000,C 180.000} C_DIS
LIN {X 57.916,Y 93.974,Z 71.556,A 180.000,B 0.000,C 180.000} C_DIS
LIN {X 57.760,Y 93.991,Z 71.552,A 180.000,B 0.000,C 180.000} C_DIS
LIN {X 57.603,Y 94.008,Z 71.549,A 180.000,B 0.000,C 180.000} C_DIS
LIN {X 57.447,Y 94.026,Z 71.546,A 180.000,B 0.000,C 180.000} C_DIS
LIN {X 57.291,Y 94.048,Z 71.543,A 180.000,B 0.000,C 180.000} C_DIS
LIN {X 57.136,Y 94.078,Z 71.540,A 180.000,B 0.000,C 180.000} C_DIS
LIN {X 56.982,Y 94.109,Z 71.537,A 180.000,B 0.000,C 180.000} C_DIS
LIN {X 56.827,Y 94.140,Z 71.534,A 180.000,B 0.000,C 180.000} C_DIS
LIN {X 56.673,Y 94.174,Z 71.532,A 180.000,B 0.000,C 180.000} C_DIS
LIN {X 56.522,Y 94.217,Z 71.529,A 180.000,B 0.000,C 180.000} C_DIS
LIN {X 56.371,Y 94.262,Z 71.527,A 180.000,B 0.000,C 180.000} C_DIS
LIN {X 56.069,Y 94.352,Z 71.522,A 180.000,B 0.000,C 180.000} C_DIS
LIN {X 55.775,Y 94.464,Z 71.518,A 180.000,B 0.000,C 180.000} C_DIS
LIN {X 55.482,Y 94.580,Z 71.514,A 180.000,B 0.000,C 180.000} C_DIS
LIN {X 55.198,Y 94.716,Z 71.511,A 180.000,B 0.000,C 180.000} C_DIS
LIN {X 54.916,Y 94.857,Z 71.508,A 180.000,B 0.000,C 180.000} C_DIS
LIN {X 54.643,Y 95.014,Z 71.505,A 180.000,B 0.000,C 180.000} C_DIS
LIN {X 54.375,Y 95.179,Z 71.503,A 180.000,B 0.000,C 180.000} C_DIS
LIN {X 54.243,Y 95.265,Z 71.503,A 180.000,B 0.000,C 180.000} C_DIS
LIN {X 54.115,Y 95.358,Z 71.502,A 180.000,B 0.000,C 180.000} C_DIS
LIN {X 53.863,Y 95.546,Z 71.501,A 180.000,B 0.000,C 180.000} C_DIS
LIN {X 53.738,Y 95.641,Z 71.500,A 180.000,B 0.000,C 180.000} C_DIS
LIN {X 53.618,Y 95.744,Z 71.500,A 180.000,B 0.000,C 180.000} C_DIS
LIN {X 53.445,Y 95.899,Z 71.500,A 180.000,B 0.000,C 180.000} C_DIS
; Cutting Move Starts
LIN {X 53.329,Y 96.003,Z 71.500,A 180.000,B 0.000,C 180.000} C_DIS
LIN {X 53.277,Y 96.050,Z 71.500,A 180.000,B 0.000,C 180.000} C_DIS
LIN {X 53.144,Y 96.181,Z 71.500,A 180.000,B 0.000,C 180.000} C_DIS
LIN {X 52.919,Y 96.421,Z 71.500,A 180.000,B 0.000,C 180.000} C_DIS
LIN {X 52.810,Y 96.539,Z 71.500,A 180.000,B 0.000,C 180.000} C_DIS
LIN {X 52.740,Y 96.619,Z 71.500,A 180.000,B 0.000,C 180.000} C_DIS
LIN {X 52.662,Y 96.718,Z 71.500,A 180.000,B 0.000,C 180.000} C_DIS
LIN {X 52.522,Y 96.897,Z 71.500,A 180.000,B 0.000,C 180.000} C_DIS
LIN {X 52.383,Y 97.075,Z 71.500,A 180.000,B 0.000,C 180.000} C_DIS
LIN {X 52.261,Y 97.254,Z 71.500,A 180.000,B 0.000,C 180.000} C_DIS
LIN {X 52.145,Y 97.433,Z 71.500,A 180.000,B 0.000,C 180.000} C_DIS
LIN {X 52.029,Y 97.612,Z 71.500,A 180.000,B 0.000,C 180.000} C_DIS
LIN {X 52.025,Y 97.618,Z 71.500,A 180.000,B 0.000,C 180.000} C_DIS
LIN {X 51.927,Y 97.790,Z 71.500,A 180.000,B 0.000,C 180.000} C_DIS
LIN {X 51.737,Y 98.148,Z 71.500,A 180.000,B 0.000,C 180.000} C_DIS
LIN {X 51.668,Y 98.287,Z 71.500,A 180.000,B 0.000,C 180.000} C_DIS
LIN {X 51.650,Y 98.327,Z 71.500,A 180.000,B 0.000,C 180.000} C_DIS
LIN {X 51.574,Y 98.505,Z 71.500,A 180.000,B 0.000,C 180.000} C_DIS
LIN {X 51.489,Y 98.708,Z 71.500,A 180.000,B 0.000,C 180.000} C_DIS
LIN {X 51.426,Y 98.863,Z 71.500,A 180.000,B 0.000,C 180.000} C_DIS
LIN {X 51.365,Y 99.042,Z 71.500,A 180.000,B 0.000,C 180.000} C_DIS
LIN {X 51.250,Y 99.399,Z 71.500,A 180.000,B 0.000,C 180.000} C_DIS
LIN {X 51.199,Y 99.578,Z 71.500,A 180.000,B 0.000,C 180.000} C_DIS
LIN {X 51.159,Y 99.757,Z 71.500,A 180.000,B 0.000,C 180.000} C_DIS
LIN {X 51.118,Y 99.936,Z 71.500,A 180.000,B 0.000,C 180.000} C_DIS
LIN {X 51.079,Y 100.114,Z 71.500,A 180.000,B 0.000,C 180.000} C_DIS
LIN {X 51.049,Y 100.293,Z 71.500,A 180.000,B 0.000,C 180.000} C_DIS
LIN {X 51.001,Y 100.651,Z 71.500,A 180.000,B 0.000,C 180.000} C_DIS
LIN {X 50.980,Y 100.829,Z 71.500,A 180.000,B 0.000,C 180.000} C_DIS
LIN {X 50.969,Y 101.008,Z 71.500,A 180.000,B 0.000,C 180.000} C_DIS
LIN {X 50.953,Y 101.385,Z 71.500,A 180.000,B 0.000,C 180.000} C_DIS
LIN {X 50.950,Y 101.545,Z 71.500,A 180.000,B 0.000,C 180.000} C_DIS
LIN {X 50.953,Y 101.615,Z 71.500,A 180.000,B 0.000,C 180.000} C_DIS
LIN {X 50.965,Y 101.902,Z 71.500,A 180.000,B 0.000,C 180.000} C_DIS
LIN {X 50.973,Y 102.081,Z 71.500,A 180.000,B 0.000,C 180.000} C_DIS
LIN {X 50.989,Y 102.260,Z 71.500,A 180.000,B 0.000,C 180.000} C_DIS
LIN {X 51.013,Y 102.438,Z 71.500,A 180.000,B 0.000,C 180.000} C_DIS
LIN {X 51.037,Y 102.617,Z 71.500,A 180.000,B 0.000,C 180.000} C_DIS
LIN {X 51.062,Y 102.796,Z 71.500,A 180.000,B 0.000,C 180.000} C_DIS
LIN {X 51.098,Y 102.975,Z 71.500,A 180.000,B 0.000,C 180.000} C_DIS
LIN {X 51.179,Y 103.332,Z 71.500,A 180.000,B 0.000,C 180.000} C_DIS
LIN {X 51.223,Y 103.511,Z 71.500,A 180.000,B 0.000,C 180.000} C_DIS
LIN {X 51.279,Y 103.690,Z 71.500,A 180.000,B 0.000,C 180.000} C_DIS
LIN {X 51.336,Y 103.869,Z 71.500,A 180.000,B 0.000,C 180.000} C_DIS
LIN {X 51.393,Y 104.047,Z 71.500,A 180.000,B 0.000,C 180.000} C_DIS
LIN {X 51.461,Y 104.226,Z 71.500,A 180.000,B 0.000,C 180.000} C_DIS
LIN {X 51.612,Y 104.584,Z 71.500,A 180.000,B 0.000,C 180.000} C_DIS
LIN {X 51.668,Y 104.713,Z 71.500,A 180.000,B 0.000,C 180.000} C_DIS
LIN {X 51.691,Y 104.762,Z 71.500,A 180.000,B 0.000,C 180.000} C_DIS
LIN {X 51.785,Y 104.941,Z 71.500,A 180.000,B 0.000,C 180.000} C_DIS
LIN {X 51.879,Y 105.120,Z 71.500,A 180.000,B 0.000,C 180.000} C_DIS
LIN {X 51.975,Y 105.299,Z 71.500,A 180.000,B 0.000,C 180.000} C_DIS
LIN {X 52.025,Y 105.382,Z 71.500,A 180.000,B 0.000,C 180.000} C_DIS
LIN {X 52.087,Y 105.477,Z 71.500,A 180.000,B 0.000,C 180.000} C_DIS
LIN {X 52.204,Y 105.658,Z 71.500,A 180.000,B 0.000,C 180.000} C_DIS
LIN {X 52.319,Y 105.835,Z 71.500,A 180.000,B 0.000,C 180.000} C_DIS
LIN {X 52.383,Y 105.925,Z 71.500,A 180.000,B 0.000,C 180.000} C_DIS
LIN {X 52.452,Y 106.014,Z 71.500,A 180.000,B 0.000,C 180.000} C_DIS
LIN {X 52.591,Y 106.193,Z 71.500,A 180.000,B 0.000,C 180.000} C_DIS
LIN {X 52.732,Y 106.371,Z 71.500,A 180.000,B 0.000,C 180.000} C_DIS
LIN {X 52.740,Y 106.381,Z 71.500,A 180.000,B 0.000,C 180.000} C_DIS
LIN {X 52.892,Y 106.550,Z 71.500,A 180.000,B 0.000,C 180.000} C_DIS
LIN {X 53.098,Y 106.770,Z 71.500,A 180.000,B 0.000,C 180.000} C_DIS
LIN {X 53.231,Y 106.908,Z 71.500,A 180.000,B 0.000,C 180.000} C_DIS
LIN {X 53.277,Y 106.950,Z 71.500,A 180.000,B 0.000,C 180.000} C_DIS
LIN {X 53.428,Y 107.086,Z 71.500,A 180.000,B 0.000,C 180.000} C_DIS
LIN {X 53.634,Y 107.271,Z 71.500,A 180.000,B 0.000,C 180.000} C_DIS
LIN {X 53.724,Y 107.347,Z 71.500,A 180.000,B 0.000,C 180.000} C_DIS
LIN {X 53.813,Y 107.417,Z 71.500,A 180.000,B 0.000,C 180.000} C_DIS
LIN {X 54.089,Y 107.623,Z 71.500,A 180.000,B 0.000,C 180.000} C_DIS
LIN {X 54.171,Y 107.684,Z 71.500,A 180.000,B 0.000,C 180.000} C_DIS
LIN {X 54.344,Y 107.802,Z 71.500,A 180.000,B 0.000,C 180.000} C_DIS
LIN {X 54.707,Y 108.025,Z 71.500,A 180.000,B 0.000,C 180.000} C_DIS
LIN {X 54.886,Y 108.128,Z 71.500,A 180.000,B 0.000,C 180.000} C_DIS
LIN {X 54.947,Y 108.159,Z 71.500,A 180.000,B 0.000,C 180.000} C_DIS
LIN {X 55.304,Y 108.338,Z 71.500,A 180.000,B 0.000,C 180.000} C_DIS
LIN {X 55.422,Y 108.394,Z 71.500,A 180.000,B 0.000,C 180.000} C_DIS
LIN {X 55.601,Y 108.467,Z 71.500,A 180.000,B 0.000,C 180.000} C_DIS
LIN {X 55.779,Y 108.538,Z 71.500,A 180.000,B 0.000,C 180.000} C_DIS
LIN {X 55.958,Y 108.608,Z 71.500,A 180.000,B 0.000,C 180.000} C_DIS
LIN {X 56.137,Y 108.669,Z 71.500,A 180.000,B 0.000,C 180.000} C_DIS
LIN {X 56.225,Y 108.695,Z 71.500,A 180.000,B 0.000,C 180.000} C_DIS
LIN {X 56.495,Y 108.775,Z 71.500,A 180.000,B 0.000,C 180.000} C_DIS
LIN {X 56.673,Y 108.826,Z 71.500,A 180.000,B 0.000,C 180.000} C_DIS
LIN {X 56.852,Y 108.865,Z 71.500,A 180.000,B 0.000,C 180.000} C_DIS
LIN {X 57.210,Y 108.937,Z 71.500,A 180.000,B 0.000,C 180.000} C_DIS
LIN {X 57.388,Y 108.967,Z 71.500,A 180.000,B 0.000,C 180.000} C_DIS
LIN {X 57.567,Y 108.988,Z 71.500,A 180.000,B 0.000,C 180.000} C_DIS
LIN {X 57.746,Y 109.008,Z 71.500,A 180.000,B 0.000,C 180.000} C_DIS
LIN {X 57.925,Y 109.027,Z 71.500,A 180.000,B 0.000,C 180.000} C_DIS
LIN {X 58.103,Y 109.038,Z 71.500,A 180.000,B 0.000,C 180.000} C_DIS
LIN {X 58.461,Y 109.046,Z 71.500,A 180.000,B 0.000,C 180.000} C_DIS
LIN {X 58.640,Y 109.049,Z 71.500,A 180.000,B 0.000,C 180.000} C_DIS
LIN {X 58.819,Y 109.041,Z 71.500,A 180.000,B 0.000,C 180.000} C_DIS
LIN {X 59.176,Y 109.017,Z 71.500,A 180.000,B 0.000,C 180.000} C_DIS
LIN {X 59.355,Y 109.001,Z 71.500,A 180.000,B 0.000,C 180.000} C_DIS
LIN {X 59.534,Y 108.975,Z 71.500,A 180.000,B 0.000,C 180.000} C_DIS
LIN {X 59.891,Y 108.919,Z 71.500,A 180.000,B 0.000,C 180.000} C_DIS
LIN {X 60.070,Y 108.884,Z 71.500,A 180.000,B 0.000,C 180.000} C_DIS
LIN {X 60.111,Y 108.874,Z 71.500,A 180.000,B 0.000,C 180.000} C_DIS
LIN {X 60.427,Y 108.796,Z 71.500,A 180.000,B 0.000,C 180.000} C_DIS
LIN {X 60.606,Y 108.750,Z 71.500,A 180.000,B 0.000,C 180.000} C_DIS
LIN {X 60.778,Y 108.695,Z 71.500,A 180.000,B 0.000,C 180.000} C_DIS
LIN {X 61.143,Y 108.570,Z 71.500,A 180.000,B 0.000,C 180.000} C_DIS
LIN {X 61.287,Y 108.517,Z 71.500,A 180.000,B 0.000,C 180.000} C_DIS
LIN {X 61.321,Y 108.503,Z 71.500,A 180.000,B 0.000,C 180.000} C_DIS
LIN {X 61.500,Y 108.424,Z 71.500,A 180.000,B 0.000,C 180.000} C_DIS
LIN {X 61.692,Y 108.338,Z 71.500,A 180.000,B 0.000,C 180.000} C_DIS
LIN {X 61.858,Y 108.262,Z 71.500,A 180.000,B 0.000,C 180.000} C_DIS
LIN {X 62.036,Y 108.167,Z 71.500,A 180.000,B 0.000,C 180.000} C_DIS
LIN {X 62.371,Y 107.980,Z 71.500,A 180.000,B 0.000,C 180.000} C_DIS
LIN {X 62.394,Y 107.967,Z 71.500,A 180.000,B 0.000,C 180.000} C_DIS
LIN {X 62.573,Y 107.855,Z 71.500,A 180.000,B 0.000,C 180.000} C_DIS
LIN {X 62.930,Y 107.612,Z 71.500,A 180.000,B 0.000,C 180.000} C_DIS
LIN {X 63.020,Y 107.548,Z 71.500,A 180.000,B 0.000,C 180.000} C_DIS
LIN {X 63.109,Y 107.478,Z 71.500,A 180.000,B 0.000,C 180.000} C_DIS
LIN {X 63.369,Y 107.265,Z 71.500,A 180.000,B 0.000,C 180.000} C_DIS
LIN {X 63.467,Y 107.185,Z 71.500,A 180.000,B 0.000,C 180.000} C_DIS
LIN {X 63.578,Y 107.086,Z 71.500,A 180.000,B 0.000,C 180.000} C_DIS
LIN {X 63.645,Y 107.021,Z 71.500,A 180.000,B 0.000,C 180.000} C_DIS
LIN {X 63.824,Y 106.847,Z 71.500,A 180.000,B 0.000,C 180.000} C_DIS
LIN {X 63.944,Y 106.729,Z 71.500,A 180.000,B 0.000,C 180.000} C_DIS
LIN {X 64.003,Y 106.669,Z 71.500,A 180.000,B 0.000,C 180.000} C_DIS
LIN {X 64.109,Y 106.550,Z 71.500,A 180.000,B 0.000,C 180.000} C_DIS
LIN {X 64.360,Y 106.256,Z 71.500,A 180.000,B 0.000,C 180.000} C_DIS
LIN {X 64.414,Y 106.193,Z 71.500,A 180.000,B 0.000,C 180.000} C_DIS
LIN {X 64.539,Y 106.026,Z 71.500,A 180.000,B 0.000,C 180.000} C_DIS
LIN {X 64.718,Y 105.776,Z 71.500,A 180.000,B 0.000,C 180.000} C_DIS
LIN {X 64.802,Y 105.656,Z 71.500,A 180.000,B 0.000,C 180.000} C_DIS
LIN {X 64.897,Y 105.507,Z 71.500,A 180.000,B 0.000,C 180.000} C_DIS
LIN {X 65.075,Y 105.203,Z 71.500,A 180.000,B 0.000,C 180.000} C_DIS
LIN {X 65.124,Y 105.120,Z 71.500,A 180.000,B 0.000,C 180.000} C_DIS
LIN {X 65.219,Y 104.941,Z 71.500,A 180.000,B 0.000,C 180.000} C_DIS
LIN {X 65.254,Y 104.866,Z 71.500,A 180.000,B 0.000,C 180.000} C_DIS
LIN {X 65.388,Y 104.584,Z 71.500,A 180.000,B 0.000,C 180.000} C_DIS
LIN {X 65.433,Y 104.488,Z 71.500,A 180.000,B 0.000,C 180.000} C_DIS
LIN {X 65.469,Y 104.405,Z 71.500,A 180.000,B 0.000,C 180.000} C_DIS
LIN {X 65.536,Y 104.226,Z 71.500,A 180.000,B 0.000,C 180.000} C_DIS
LIN {X 65.612,Y 104.022,Z 71.500,A 180.000,B 0.000,C 180.000} C_DIS
LIN {X 65.668,Y 103.869,Z 71.500,A 180.000,B 0.000,C 180.000} C_DIS
LIN {X 65.724,Y 103.690,Z 71.500,A 180.000,B 0.000,C 180.000} C_DIS
LIN {X 65.821,Y 103.332,Z 71.500,A 180.000,B 0.000,C 180.000} C_DIS
LIN {X 65.867,Y 103.153,Z 71.500,A 180.000,B 0.000,C 180.000} C_DIS
LIN {X 65.901,Y 102.975,Z 71.500,A 180.000,B 0.000,C 180.000} C_DIS
LIN {X 65.965,Y 102.617,Z 71.500,A 180.000,B 0.000,C 180.000} C_DIS
LIN {X 65.969,Y 102.592,Z 71.500,A 180.000,B 0.000,C 180.000} C_DIS
LIN {X 65.991,Y 102.438,Z 71.500,A 180.000,B 0.000,C 180.000} C_DIS
LIN {X 66.007,Y 102.260,Z 71.500,A 180.000,B 0.000,C 180.000} C_DIS
LIN {X 66.023,Y 102.081,Z 71.500,A 180.000,B 0.000,C 180.000} C_DIS
LIN {X 66.039,Y 101.902,Z 71.500,A 180.000,B 0.000,C 180.000} C_DIS
LIN {X 66.045,Y 101.723,Z 71.500,A 180.000,B 0.000,C 180.000} C_DIS
LIN {X 66.045,Y 101.366,Z 71.500,A 180.000,B 0.000,C 180.000} C_DIS
LIN {X 66.043,Y 101.187,Z 71.500,A 180.000,B 0.000,C 180.000} C_DIS
LIN {X 66.031,Y 101.008,Z 71.500,A 180.000,B 0.000,C 180.000} C_DIS
LIN {X 65.999,Y 100.651,Z 71.500,A 180.000,B 0.000,C 180.000} C_DIS
LIN {X 65.980,Y 100.472,Z 71.500,A 180.000,B 0.000,C 180.000} C_DIS
LIN {X 65.969,Y 100.408,Z 71.500,A 180.000,B 0.000,C 180.000} C_DIS
LIN {X 65.949,Y 100.293,Z 71.500,A 180.000,B 0.000,C 180.000} C_DIS
LIN {X 65.917,Y 100.114,Z 71.500,A 180.000,B 0.000,C 180.000} C_DIS
LIN {X 65.885,Y 99.936,Z 71.500,A 180.000,B 0.000,C 180.000} C_DIS
LIN {X 65.845,Y 99.757,Z 71.500,A 180.000,B 0.000,C 180.000} C_DIS
LIN {X 65.796,Y 99.578,Z 71.500,A 180.000,B 0.000,C 180.000} C_DIS
LIN {X 65.748,Y 99.399,Z 71.500,A 180.000,B 0.000,C 180.000} C_DIS
LIN {X 65.698,Y 99.221,Z 71.500,A 180.000,B 0.000,C 180.000} C_DIS
LIN {X 65.635,Y 99.042,Z 71.500,A 180.000,B 0.000,C 180.000} C_DIS
LIN {X 65.503,Y 98.684,Z 71.500,A 180.000,B 0.000,C 180.000} C_DIS
LIN {X 65.433,Y 98.512,Z 71.500,A 180.000,B 0.000,C 180.000} C_DIS
LIN {X 65.430,Y 98.505,Z 71.500,A 180.000,B 0.000,C 180.000} C_DIS
LIN {X 65.346,Y 98.327,Z 71.500,A 180.000,B 0.000,C 180.000} C_DIS
LIN {X 65.254,Y 98.134,Z 71.500,A 180.000,B 0.000,C 180.000} C_DIS
LIN {X 65.174,Y 97.969,Z 71.500,A 180.000,B 0.000,C 180.000} C_DIS
LIN {X 65.075,Y 97.797,Z 71.500,A 180.000,B 0.000,C 180.000} C_DIS
LIN {X 64.897,Y 97.493,Z 71.500,A 180.000,B 0.000,C 180.000} C_DIS
LIN {X 64.861,Y 97.433,Z 71.500,A 180.000,B 0.000,C 180.000} C_DIS
LIN {X 64.739,Y 97.254,Z 71.500,A 180.000,B 0.000,C 180.000} C_DIS
LIN {X 64.539,Y 96.974,Z 71.500,A 180.000,B 0.000,C 180.000} C_DIS
LIN {X 64.484,Y 96.897,Z 71.500,A 180.000,B 0.000,C 180.000} C_DIS
LIN {X 64.360,Y 96.744,Z 71.500,A 180.000,B 0.000,C 180.000} C_DIS
LIN {X 64.182,Y 96.535,Z 71.500,A 180.000,B 0.000,C 180.000} C_DIS
LIN {X 64.030,Y 96.360,Z 71.500,A 180.000,B 0.000,C 180.000} C_DIS
LIN {X 64.003,Y 96.331,Z 71.500,A 180.000,B 0.000,C 180.000} C_DIS
LIN {X 63.853,Y 96.181,Z 71.500,A 180.000,B 0.000,C 180.000} C_DIS
LIN {X 63.645,Y 95.979,Z 71.500,A 180.000,B 0.000,C 180.000} C_DIS
LIN {X 63.477,Y 95.824,Z 71.500,A 180.000,B 0.000,C 180.000} C_DIS
LIN {X 63.467,Y 95.815,Z 71.500,A 180.000,B 0.000,C 180.000} C_DIS
LIN {X 63.288,Y 95.669,Z 71.500,A 180.000,B 0.000,C 180.000} C_DIS
LIN {X 63.109,Y 95.522,Z 71.500,A 180.000,B 0.000,C 180.000} C_DIS
LIN {X 63.038,Y 95.466,Z 71.500,A 180.000,B 0.000,C 180.000} C_DIS
LIN {X 62.930,Y 95.388,Z 71.500,A 180.000,B 0.000,C 180.000} C_DIS
LIN {X 62.573,Y 95.145,Z 71.500,A 180.000,B 0.000,C 180.000} C_DIS
LIN {X 62.518,Y 95.109,Z 71.500,A 180.000,B 0.000,C 180.000} C_DIS
LIN {X 62.394,Y 95.033,Z 71.500,A 180.000,B 0.000,C 180.000} C_DIS
LIN {X 62.210,Y 94.930,Z 71.500,A 180.000,B 0.000,C 180.000} C_DIS
LIN {X 62.036,Y 94.833,Z 71.500,A 180.000,B 0.000,C 180.000} C_DIS
LIN {X 61.885,Y 94.751,Z 71.500,A 180.000,B 0.000,C 180.000} C_DIS
LIN {X 61.858,Y 94.738,Z 71.500,A 180.000,B 0.000,C 180.000} C_DIS
LIN {X 61.679,Y 94.656,Z 71.500,A 180.000,B 0.000,C 180.000} C_DIS
LIN {X 61.491,Y 94.573,Z 71.500,A 180.000,B 0.000,C 180.000} C_DIS
LIN {X 61.321,Y 94.497,Z 71.500,A 180.000,B 0.000,C 180.000} C_DIS
LIN {X 61.143,Y 94.430,Z 71.500,A 180.000,B 0.000,C 180.000} C_DIS
LIN {X 60.785,Y 94.307,Z 71.500,A 180.000,B 0.000,C 180.000} C_DIS
LIN {X 60.606,Y 94.250,Z 71.500,A 180.000,B 0.000,C 180.000} C_DIS
LIN {X 60.470,Y 94.215,Z 71.500,A 180.000,B 0.000,C 180.000} C_DIS
LIN {X 60.249,Y 94.160,Z 71.500,A 180.000,B 0.000,C 180.000} C_DIS
LIN {X 60.070,Y 94.116,Z 71.500,A 180.000,B 0.000,C 180.000} C_DIS
LIN {X 59.891,Y 94.081,Z 71.500,A 180.000,B 0.000,C 180.000} C_DIS
LIN {X 59.534,Y 94.025,Z 71.500,A 180.000,B 0.000,C 180.000} C_DIS
LIN {X 59.355,Y 93.999,Z 71.500,A 180.000,B 0.000,C 180.000} C_DIS
LIN {X 59.176,Y 93.983,Z 71.500,A 180.000,B 0.000,C 180.000} C_DIS
LIN {X 58.819,Y 93.959,Z 71.500,A 180.000,B 0.000,C 180.000} C_DIS
LIN {X 58.640,Y 93.951,Z 71.500,A 180.000,B 0.000,C 180.000} C_DIS
LIN {X 58.461,Y 93.954,Z 71.500,A 180.000,B 0.000,C 180.000} C_DIS
LIN {X 58.103,Y 93.962,Z 71.500,A 180.000,B 0.000,C 180.000} C_DIS
LIN {X 57.925,Y 93.973,Z 71.500,A 180.000,B 0.000,C 180.000} C_DIS
LIN {X 57.746,Y 93.992,Z 71.500,A 180.000,B 0.000,C 180.000} C_DIS
LIN {X 57.567,Y 94.012,Z 71.500,A 180.000,B 0.000,C 180.000} C_DIS
LIN {X 57.388,Y 94.033,Z 71.500,A 180.000,B 0.000,C 180.000} C_DIS
LIN {X 57.363,Y 94.036,Z 71.500,A 180.000,B 0.000,C 180.000} C_DIS
LIN {X 57.210,Y 94.063,Z 71.500,A 180.000,B 0.000,C 180.000} C_DIS
LIN {X 56.852,Y 94.135,Z 71.500,A 180.000,B 0.000,C 180.000} C_DIS
LIN {X 56.673,Y 94.174,Z 71.500,A 180.000,B 0.000,C 180.000} C_DIS
LIN {X 56.528,Y 94.215,Z 71.500,A 180.000,B 0.000,C 180.000} C_DIS
LIN {X 56.316,Y 94.278,Z 71.500,A 180.000,B 0.000,C 180.000} C_DIS
LIN {X 56.137,Y 94.331,Z 71.500,A 180.000,B 0.000,C 180.000} C_DIS
LIN {X 55.958,Y 94.392,Z 71.500,A 180.000,B 0.000,C 180.000} C_DIS
LIN {X 55.953,Y 94.394,Z 71.500,A 180.000,B 0.000,C 180.000} C_DIS
LIN {X 55.779,Y 94.462,Z 71.500,A 180.000,B 0.000,C 180.000} C_DIS
LIN {X 55.601,Y 94.533,Z 71.500,A 180.000,B 0.000,C 180.000} C_DIS
LIN {X 55.501,Y 94.573,Z 71.500,A 180.000,B 0.000,C 180.000} C_DIS
LIN {X 55.422,Y 94.606,Z 71.500,A 180.000,B 0.000,C 180.000} C_DIS
LIN {X 55.243,Y 94.693,Z 71.500,A 180.000,B 0.000,C 180.000} C_DIS
LIN {X 55.064,Y 94.782,Z 71.500,A 180.000,B 0.000,C 180.000} C_DIS
LIN {X 54.886,Y 94.872,Z 71.500,A 180.000,B 0.000,C 180.000} C_DIS
LIN {X 54.781,Y 94.930,Z 71.500,A 180.000,B 0.000,C 180.000} C_DIS
LIN {X 54.707,Y 94.975,Z 71.500,A 180.000,B 0.000,C 180.000} C_DIS
LIN {X 54.349,Y 95.195,Z 71.500,A 180.000,B 0.000,C 180.000} C_DIS
LIN {X 54.210,Y 95.288,Z 71.500,A 180.000,B 0.000,C 180.000} C_DIS
LIN {X 54.171,Y 95.316,Z 71.500,A 180.000,B 0.000,C 180.000} C_DIS
LIN {X 53.970,Y 95.466,Z 71.500,A 180.000,B 0.000,C 180.000} C_DIS
LIN {X 53.813,Y 95.583,Z 71.500,A 180.000,B 0.000,C 180.000} C_DIS
LIN {X 53.733,Y 95.645,Z 71.500,A 180.000,B 0.000,C 180.000} C_DIS
LIN {X 53.634,Y 95.729,Z 71.500,A 180.000,B 0.000,C 180.000} C_DIS
LIN {X 53.445,Y 95.899,Z 71.500,A 180.000,B 0.000,C 180.000} C_DIS
; Link Move Starts
LIN {X 53.212,Y 96.111,Z 71.500,A 180.000,B 0.000,C 180.000} C_DIS
LIN {X 52.995,Y 96.340,Z 71.499,A 180.000,B 0.000,C 180.000} C_DIS
LIN {X 52.781,Y 96.571,Z 71.498,A 180.000,B 0.000,C 180.000} C_DIS
LIN {X 52.584,Y 96.817,Z 71.496,A 180.000,B 0.000,C 180.000} C_DIS
LIN {X 52.391,Y 97.065,Z 71.494,A 180.000,B 0.000,C 180.000} C_DIS
LIN {X 52.214,Y 97.326,Z 71.491,A 180.000,B 0.000,C 180.000} C_DIS
LIN {X 52.043,Y 97.590,Z 71.488,A 180.000,B 0.000,C 180.000} C_DIS
LIN {X 51.888,Y 97.864,Z 71.485,A 180.000,B 0.000,C 180.000} C_DIS
LIN {X 51.740,Y 98.143,Z 71.481,A 180.000,B 0.000,C 180.000} C_DIS
LIN {X 51.669,Y 98.283,Z 71.479,A 180.000,B 0.000,C 180.000} C_DIS
LIN {X 51.607,Y 98.428,Z 71.477,A 180.000,B 0.000,C 180.000} C_DIS
LIN {X 51.485,Y 98.718,Z 71.472,A 180.000,B 0.000,C 180.000} C_DIS
LIN {X 51.425,Y 98.864,Z 71.469,A 180.000,B 0.000,C 180.000} C_DIS
LIN {X 51.374,Y 99.013,Z 71.467,A 180.000,B 0.000,C 180.000} C_DIS
LIN {X 51.326,Y 99.163,Z 71.464,A 180.000,B 0.000,C 180.000} C_DIS
LIN {X 51.278,Y 99.313,Z 71.461,A 180.000,B 0.000,C 180.000} C_DIS
LIN {X 51.230,Y 99.463,Z 71.459,A 180.000,B 0.000,C 180.000} C_DIS
LIN {X 51.190,Y 99.616,Z 71.456,A 180.000,B 0.000,C 180.000} C_DIS
LIN {X 51.156,Y 99.769,Z 71.452,A 180.000,B 0.000,C 180.000} C_DIS
LIN {X 51.121,Y 99.923,Z 71.449,A 180.000,B 0.000,C 180.000} C_DIS
LIN {X 51.087,Y 100.077,Z 71.446,A 180.000,B 0.000,C 180.000} C_DIS
LIN {X 51.058,Y 100.231,Z 71.443,A 180.000,B 0.000,C 180.000} C_DIS
LIN {X 51.037,Y 100.387,Z 71.439,A 180.000,B 0.000,C 180.000} C_DIS
LIN {X 51.016,Y 100.544,Z 71.436,A 180.000,B 0.000,C 180.000} C_DIS
LIN {X 50.995,Y 100.700,Z 71.432,A 180.000,B 0.000,C 180.000} C_DIS
LIN {X 50.978,Y 100.856,Z 71.428,A 180.000,B 0.000,C 180.000} C_DIS
LIN {X 50.969,Y 101.014,Z 71.425,A 180.000,B 0.000,C 180.000} C_DIS
LIN {X 50.962,Y 101.171,Z 71.421,A 180.000,B 0.000,C 180.000} C_DIS
LIN {X 50.955,Y 101.328,Z 71.417,A 180.000,B 0.000,C 180.000} C_DIS
LIN {X 50.950,Y 101.486,Z 71.413,A 180.000,B 0.000,C 180.000} C_DIS
LIN {X 50.954,Y 101.643,Z 71.409,A 180.000,B 0.000,C 180.000} C_DIS
LIN {X 50.961,Y 101.800,Z 71.405,A 180.000,B 0.000,C 180.000} C_DIS
LIN {X 50.968,Y 101.958,Z 71.400,A 180.000,B 0.000,C 180.000} C_DIS
LIN {X 50.975,Y 102.115,Z 71.396,A 180.000,B 0.000,C 180.000} C_DIS
LIN {X 50.991,Y 102.272,Z 71.392,A 180.000,B 0.000,C 180.000} C_DIS
LIN {X 51.012,Y 102.428,Z 71.387,A 180.000,B 0.000,C 180.000} C_DIS
LIN {X 51.033,Y 102.584,Z 71.383,A 180.000,B 0.000,C 180.000} C_DIS
LIN {X 51.054,Y 102.740,Z 71.378,A 180.000,B 0.000,C 180.000} C_DIS
LIN {X 51.081,Y 102.895,Z 71.373,A 180.000,B 0.000,C 180.000} C_DIS
LIN {X 51.115,Y 103.049,Z 71.369,A 180.000,B 0.000,C 180.000} C_DIS
LIN {X 51.149,Y 103.203,Z 71.364,A 180.000,B 0.000,C 180.000} C_DIS
LIN {X 51.184,Y 103.356,Z 71.359,A 180.000,B 0.000,C 180.000} C_DIS
LIN {X 51.222,Y 103.509,Z 71.354,A 180.000,B 0.000,C 180.000} C_DIS
LIN {X 51.245,Y 103.585,Z 71.351,A 180.000,B 0.000,C 180.000} C_DIS
LIN {X 51.269,Y 103.660,Z 71.349,A 180.000,B 0.000,C 180.000} C_DIS
LIN {X 51.293,Y 103.735,Z 71.346,A 180.000,B 0.000,C 180.000} C_DIS
LIN {X 51.317,Y 103.810,Z 71.344,A 180.000,B 0.000,C 180.000} C_DIS
LIN {X 51.341,Y 103.885,Z 71.341,A 180.000,B 0.000,C 180.000} C_DIS
LIN {X 51.365,Y 103.960,Z 71.339,A 180.000,B 0.000,C 180.000} C_DIS
LIN {X 51.389,Y 104.035,Z 71.336,A 180.000,B 0.000,C 180.000} C_DIS
LIN {X 51.415,Y 104.109,Z 71.333,A 180.000,B 0.000,C 180.000} C_DIS
LIN {X 51.443,Y 104.182,Z 71.331,A 180.000,B 0.000,C 180.000} C_DIS
LIN {X 51.474,Y 104.255,Z 71.328,A 180.000,B 0.000,C 180.000} C_DIS
LIN {X 51.535,Y 104.400,Z 71.323,A 180.000,B 0.000,C 180.000} C_DIS
LIN {X 51.596,Y 104.546,Z 71.317,A 180.000,B 0.000,C 180.000} C_DIS
LIN {X 51.626,Y 104.618,Z 71.315,A 180.000,B 0.000,C 180.000} C_DIS
LIN {X 51.658,Y 104.690,Z 71.312,A 180.000,B 0.000,C 180.000} C_DIS
LIN {X 51.691,Y 104.762,Z 71.309,A 180.000,B 0.000,C 180.000} C_DIS
LIN {X 51.727,Y 104.832,Z 71.307,A 180.000,B 0.000,C 180.000} C_DIS
LIN {X 51.800,Y 104.971,Z 71.301,A 180.000,B 0.000,C 180.000} C_DIS
LIN {X 51.911,Y 105.180,Z 71.293,A 180.000,B 0.000,C 180.000} C_DIS
LIN {X 51.948,Y 105.249,Z 71.290,A 180.000,B 0.000,C 180.000} C_DIS
LIN {X 51.987,Y 105.318,Z 71.287,A 180.000,B 0.000,C 180.000} C_DIS
LIN {X 52.027,Y 105.385,Z 71.285,A 180.000,B 0.000,C 180.000} C_DIS
LIN {X 52.070,Y 105.452,Z 71.282,A 180.000,B 0.000,C 180.000} C_DIS
LIN {X 52.156,Y 105.584,Z 71.276,A 180.000,B 0.000,C 180.000} C_DIS
LIN {X 52.198,Y 105.650,Z 71.274,A 180.000,B 0.000,C 180.000} C_DIS
LIN {X 52.284,Y 105.782,Z 71.268,A 180.000,B 0.000,C 180.000} C_DIS
LIN {X 52.328,Y 105.848,Z 71.265,A 180.000,B 0.000,C 180.000} C_DIS
LIN {X 52.373,Y 105.912,Z 71.263,A 180.000,B 0.000,C 180.000} C_DIS
LIN {X 52.421,Y 105.975,Z 71.260,A 180.000,B 0.000,C 180.000} C_DIS
LIN {X 52.518,Y 106.099,Z 71.254,A 180.000,B 0.000,C 180.000} C_DIS
LIN {X 52.566,Y 106.161,Z 71.252,A 180.000,B 0.000,C 180.000} C_DIS
LIN {X 52.664,Y 106.285,Z 71.246,A 180.000,B 0.000,C 180.000} C_DIS
LIN {X 52.712,Y 106.347,Z 71.243,A 180.000,B 0.000,C 180.000} C_DIS
LIN {X 52.762,Y 106.407,Z 71.241,A 180.000,B 0.000,C 180.000} C_DIS
LIN {X 52.814,Y 106.466,Z 71.238,A 180.000,B 0.000,C 180.000} C_DIS
LIN {X 52.868,Y 106.524,Z 71.235,A 180.000,B 0.000,C 180.000} C_DIS
LIN {X 53.029,Y 106.697,Z 71.227,A 180.000,B 0.000,C 180.000} C_DIS
LIN {X 53.137,Y 106.812,Z 71.221,A 180.000,B 0.000,C 180.000} C_DIS
LIN {X 53.192,Y 106.868,Z 71.219,A 180.000,B 0.000,C 180.000} C_DIS
LIN {X 53.248,Y 106.924,Z 71.216,A 180.000,B 0.000,C 180.000} C_DIS
LIN {X 53.306,Y 106.977,Z 71.213,A 180.000,B 0.000,C 180.000} C_DIS
LIN {X 53.599,Y 107.239,Z 71.199,A 180.000,B 0.000,C 180.000} C_DIS
LIN {X 53.658,Y 107.292,Z 71.197,A 180.000,B 0.000,C 180.000} C_DIS
LIN {X 53.718,Y 107.343,Z 71.194,A 180.000,B 0.000,C 180.000} C_DIS
LIN {X 53.780,Y 107.392,Z 71.191,A 180.000,B 0.000,C 180.000} C_DIS
LIN {X 53.843,Y 107.439,Z 71.188,A 180.000,B 0.000,C 180.000} C_DIS
LIN {X 53.906,Y 107.486,Z 71.186,A 180.000,B 0.000,C 180.000} C_DIS
LIN {X 54.032,Y 107.580,Z 71.180,A 180.000,B 0.000,C 180.000} C_DIS
LIN {X 54.158,Y 107.675,Z 71.175,A 180.000,B 0.000,C 180.000} C_DIS
LIN {X 54.222,Y 107.721,Z 71.172,A 180.000,B 0.000,C 180.000} C_DIS
LIN {X 54.287,Y 107.765,Z 71.169,A 180.000,B 0.000,C 180.000} C_DIS
LIN {X 54.354,Y 107.807,Z 71.166,A 180.000,B 0.000,C 180.000} C_DIS
LIN {X 54.488,Y 107.890,Z 71.161,A 180.000,B 0.000,C 180.000} C_DIS
LIN {X 54.689,Y 108.014,Z 71.153,A 180.000,B 0.000,C 180.000} C_DIS
LIN {X 54.756,Y 108.055,Z 71.150,A 180.000,B 0.000,C 180.000} C_DIS
LIN {X 54.824,Y 108.095,Z 71.147,A 180.000,B 0.000,C 180.000} C_DIS
LIN {X 54.894,Y 108.132,Z 71.144,A 180.000,B 0.000,C 180.000} C_DIS
LIN {X 54.964,Y 108.167,Z 71.142,A 180.000,B 0.000,C 180.000} C_DIS
LIN {X 55.175,Y 108.273,Z 71.133,A 180.000,B 0.000,C 180.000} C_DIS
LIN {X 55.316,Y 108.344,Z 71.128,A 180.000,B 0.000,C 180.000} C_DIS
LIN {X 55.387,Y 108.378,Z 71.125,A 180.000,B 0.000,C 180.000} C_DIS
LIN {X 55.459,Y 108.410,Z 71.122,A 180.000,B 0.000,C 180.000} C_DIS
LIN {X 55.532,Y 108.440,Z 71.120,A 180.000,B 0.000,C 180.000} C_DIS
LIN {X 55.751,Y 108.527,Z 71.111,A 180.000,B 0.000,C 180.000} C_DIS
LIN {X 55.898,Y 108.584,Z 71.106,A 180.000,B 0.000,C 180.000} C_DIS
LIN {X 55.971,Y 108.613,Z 71.103,A 180.000,B 0.000,C 180.000} C_DIS
LIN {X 56.045,Y 108.640,Z 71.100,A 180.000,B 0.000,C 180.000} C_DIS
LIN {X 56.120,Y 108.664,Z 71.098,A 180.000,B 0.000,C 180.000} C_DIS
LIN {X 56.196,Y 108.687,Z 71.095,A 180.000,B 0.000,C 180.000} C_DIS
LIN {X 56.573,Y 108.798,Z 71.081,A 180.000,B 0.000,C 180.000} C_DIS
LIN {X 56.649,Y 108.819,Z 71.078,A 180.000,B 0.000,C 180.000} C_DIS
LIN {X 56.726,Y 108.838,Z 71.076,A 180.000,B 0.000,C 180.000} C_DIS
LIN {X 56.803,Y 108.855,Z 71.073,A 180.000,B 0.000,C 180.000} C_DIS
LIN {X 57.189,Y 108.933,Z 71.059,A 180.000,B 0.000,C 180.000} C_DIS
LIN {X 57.266,Y 108.948,Z 71.056,A 180.000,B 0.000,C 180.000} C_DIS
LIN {X 57.344,Y 108.961,Z 71.054,A 180.000,B 0.000,C 180.000} C_DIS
LIN {X 57.422,Y 108.972,Z 71.051,A 180.000,B 0.000,C 180.000} C_DIS
LIN {X 57.500,Y 108.980,Z 71.048,A 180.000,B 0.000,C 180.000} C_DIS
LIN {X 57.891,Y 109.024,Z 71.034,A 180.000,B 0.000,C 180.000} C_DIS
LIN {X 57.970,Y 109.031,Z 71.032,A 180.000,B 0.000,C 180.000} C_DIS
LIN {X 58.048,Y 109.036,Z 71.029,A 180.000,B 0.000,C 180.000} C_DIS
LIN {X 58.127,Y 109.039,Z 71.026,A 180.000,B 0.000,C 180.000} C_DIS
LIN {X 58.521,Y 109.047,Z 71.012,A 180.000,B 0.000,C 180.000} C_DIS
LIN {X 58.599,Y 109.049,Z 71.010,A 180.000,B 0.000,C 180.000} C_DIS
LIN {X 58.678,Y 109.048,Z 71.007,A 180.000,B 0.000,C 180.000} C_DIS
LIN {X 58.757,Y 109.045,Z 71.004,A 180.000,B 0.000,C 180.000} C_DIS
LIN {X 58.835,Y 109.039,Z 71.001,A 180.000,B 0.000,C 180.000} C_DIS
LIN {X 59.228,Y 109.013,Z 70.988,A 180.000,B 0.000,C 180.000} C_DIS
LIN {X 59.307,Y 109.007,Z 70.985,A 180.000,B 0.000,C 180.000} C_DIS
LIN {X 59.385,Y 108.998,Z 70.982,A 180.000,B 0.000,C 180.000} C_DIS
LIN {X 59.463,Y 108.986,Z 70.979,A 180.000,B 0.000,C 180.000} C_DIS
LIN {X 59.852,Y 108.925,Z 70.966,A 180.000,B 0.000,C 180.000} C_DIS
LIN {X 59.930,Y 108.913,Z 70.963,A 180.000,B 0.000,C 180.000} C_DIS
LIN {X 60.007,Y 108.898,Z 70.960,A 180.000,B 0.000,C 180.000} C_DIS
LIN {X 60.084,Y 108.881,Z 70.957,A 180.000,B 0.000,C 180.000} C_DIS
LIN {X 60.160,Y 108.862,Z 70.955,A 180.000,B 0.000,C 180.000} C_DIS
LIN {X 60.466,Y 108.786,Z 70.944,A 180.000,B 0.000,C 180.000} C_DIS
LIN {X 60.542,Y 108.767,Z 70.941,A 180.000,B 0.000,C 180.000} C_DIS
LIN {X 60.619,Y 108.747,Z 70.938,A 180.000,B 0.000,C 180.000} C_DIS
LIN {X 60.694,Y 108.724,Z 70.935,A 180.000,B 0.000,C 180.000} C_DIS
LIN {X 60.769,Y 108.699,Z 70.933,A 180.000,B 0.000,C 180.000} C_DIS
LIN {X 61.141,Y 108.570,Z 70.919,A 180.000,B 0.000,C 180.000} C_DIS
LIN {X 61.215,Y 108.544,Z 70.916,A 180.000,B 0.000,C 180.000} C_DIS
LIN {X 61.289,Y 108.516,Z 70.913,A 180.000,B 0.000,C 180.000} C_DIS
LIN {X 61.361,Y 108.486,Z 70.911,A 180.000,B 0.000,C 180.000} C_DIS
LIN {X 61.433,Y 108.453,Z 70.908,A 180.000,B 0.000,C 180.000} C_DIS
LIN {X 61.721,Y 108.325,Z 70.897,A 180.000,B 0.000,C 180.000} C_DIS
LIN {X 61.793,Y 108.293,Z 70.894,A 180.000,B 0.000,C 180.000} C_DIS
LIN {X 61.864,Y 108.259,Z 70.891,A 180.000,B 0.000,C 180.000} C_DIS
LIN {X 61.934,Y 108.223,Z 70.889,A 180.000,B 0.000,C 180.000} C_DIS
LIN {X 62.003,Y 108.185,Z 70.886,A 180.000,B 0.000,C 180.000} C_DIS
LIN {X 62.347,Y 107.994,Z 70.872,A 180.000,B 0.000,C 180.000} C_DIS
LIN {X 62.415,Y 107.955,Z 70.869,A 180.000,B 0.000,C 180.000} C_DIS
LIN {X 62.483,Y 107.914,Z 70.867,A 180.000,B 0.000,C 180.000} C_DIS
LIN {X 62.549,Y 107.871,Z 70.864,A 180.000,B 0.000,C 180.000} C_DIS
LIN {X 62.614,Y 107.827,Z 70.861,A 180.000,B 0.000,C 180.000} C_DIS
LIN {X 62.874,Y 107.650,Z 70.850,A 180.000,B 0.000,C 180.000} C_DIS
LIN {X 62.940,Y 107.605,Z 70.847,A 180.000,B 0.000,C 180.000} C_DIS
LIN {X 63.004,Y 107.560,Z 70.845,A 180.000,B 0.000,C 180.000} C_DIS
LIN {X 63.066,Y 107.512,Z 70.842,A 180.000,B 0.000,C 180.000} C_DIS
LIN {X 63.128,Y 107.462,Z 70.839,A 180.000,B 0.000,C 180.000} C_DIS
LIN {X 63.432,Y 107.213,Z 70.825,A 180.000,B 0.000,C 180.000} C_DIS
LIN {X 63.493,Y 107.163,Z 70.823,A 180.000,B 0.000,C 180.000} C_DIS
LIN {X 63.552,Y 107.111,Z 70.820,A 180.000,B 0.000,C 180.000} C_DIS
LIN {X 63.609,Y 107.057,Z 70.817,A 180.000,B 0.000,C 180.000} C_DIS
LIN {X 63.666,Y 107.002,Z 70.814,A 180.000,B 0.000,C 180.000} C_DIS
LIN {X 63.722,Y 106.947,Z 70.812,A 180.000,B 0.000,C 180.000} C_DIS
LIN {X 63.835,Y 106.836,Z 70.806,A 180.000,B 0.000,C 180.000} C_DIS
LIN {X 63.891,Y 106.781,Z 70.803,A 180.000,B 0.000,C 180.000} C_DIS
LIN {X 63.947,Y 106.726,Z 70.801,A 180.000,B 0.000,C 180.000} C_DIS
LIN {X 64.002,Y 106.670,Z 70.798,A 180.000,B 0.000,C 180.000} C_DIS
LIN {X 64.055,Y 106.612,Z 70.795,A 180.000,B 0.000,C 180.000} C_DIS
LIN {X 64.107,Y 106.552,Z 70.792,A 180.000,B 0.000,C 180.000} C_DIS
LIN {X 64.158,Y 106.493,Z 70.790,A 180.000,B 0.000,C 180.000} C_DIS
LIN {X 64.261,Y 106.373,Z 70.784,A 180.000,B 0.000,C 180.000} C_DIS
LIN {X 64.363,Y 106.253,Z 70.779,A 180.000,B 0.000,C 180.000} C_DIS
LIN {X 64.414,Y 106.193,Z 70.776,A 180.000,B 0.000,C 180.000} C_DIS
LIN {X 64.463,Y 106.131,Z 70.773,A 180.000,B 0.000,C 180.000} C_DIS
LIN {X 64.510,Y 106.068,Z 70.770,A 180.000,B 0.000,C 180.000} C_DIS
LIN {X 64.555,Y 106.004,Z 70.768,A 180.000,B 0.000,C 180.000} C_DIS
LIN {X 64.647,Y 105.876,Z 70.762,A 180.000,B 0.000,C 180.000} C_DIS
LIN {X 64.738,Y 105.747,Z 70.757,A 180.000,B 0.000,C 180.000} C_DIS
LIN {X 64.784,Y 105.683,Z 70.754,A 180.000,B 0.000,C 180.000} C_DIS
LIN {X 64.828,Y 105.618,Z 70.751,A 180.000,B 0.000,C 180.000} C_DIS
LIN {X 64.870,Y 105.551,Z 70.748,A 180.000,B 0.000,C 180.000} C_DIS
LIN {X 64.910,Y 105.484,Z 70.746,A 180.000,B 0.000,C 180.000} C_DIS
LIN {X 64.990,Y 105.348,Z 70.740,A 180.000,B 0.000,C 180.000} C_DIS
LIN {X 65.110,Y 105.144,Z 70.732,A 180.000,B 0.000,C 180.000} C_DIS
LIN {X 65.149,Y 105.076,Z 70.729,A 180.000,B 0.000,C 180.000} C_DIS
LIN {X 65.186,Y 105.007,Z 70.726,A 180.000,B 0.000,C 180.000} C_DIS
LIN {X 65.221,Y 104.936,Z 70.724,A 180.000,B 0.000,C 180.000} C_DIS
LIN {X 65.289,Y 104.794,Z 70.718,A 180.000,B 0.000,C 180.000} C_DIS
LIN {X 65.390,Y 104.580,Z 70.710,A 180.000,B 0.000,C 180.000} C_DIS
LIN {X 65.423,Y 104.509,Z 70.707,A 180.000,B 0.000,C 180.000} C_DIS
LIN {X 65.455,Y 104.437,Z 70.704,A 180.000,B 0.000,C 180.000} C_DIS
LIN {X 65.485,Y 104.364,Z 70.702,A 180.000,B 0.000,C 180.000} C_DIS
LIN {X 65.513,Y 104.290,Z 70.699,A 180.000,B 0.000,C 180.000} C_DIS
LIN {X 65.567,Y 104.142,Z 70.693,A 180.000,B 0.000,C 180.000} C_DIS
LIN {X 65.649,Y 103.921,Z 70.685,A 180.000,B 0.000,C 180.000} C_DIS
LIN {X 65.676,Y 103.847,Z 70.682,A 180.000,B 0.000,C 180.000} C_DIS
LIN {X 65.700,Y 103.772,Z 70.680,A 180.000,B 0.000,C 180.000} C_DIS
LIN {X 65.722,Y 103.696,Z 70.677,A 180.000,B 0.000,C 180.000} C_DIS
LIN {X 65.763,Y 103.544,Z 70.672,A 180.000,B 0.000,C 180.000} C_DIS
LIN {X 65.804,Y 103.392,Z 70.666,A 180.000,B 0.000,C 180.000} C_DIS
LIN {X 65.825,Y 103.316,Z 70.664,A 180.000,B 0.000,C 180.000} C_DIS
LIN {X 65.846,Y 103.240,Z 70.661,A 180.000,B 0.000,C 180.000} C_DIS
LIN {X 65.864,Y 103.164,Z 70.659,A 180.000,B 0.000,C 180.000} C_DIS
LIN {X 65.881,Y 103.087,Z 70.656,A 180.000,B 0.000,C 180.000} C_DIS
LIN {X 65.895,Y 103.009,Z 70.654,A 180.000,B 0.000,C 180.000} C_DIS
LIN {X 65.909,Y 102.932,Z 70.651,A 180.000,B 0.000,C 180.000} C_DIS
LIN {X 65.923,Y 102.854,Z 70.649,A 180.000,B 0.000,C 180.000} C_DIS
LIN {X 65.950,Y 102.699,Z 70.644,A 180.000,B 0.000,C 180.000} C_DIS
LIN {X 65.977,Y 102.544,Z 70.639,A 180.000,B 0.000,C 180.000} C_DIS
LIN {X 65.996,Y 102.387,Z 70.634,A 180.000,B 0.000,C 180.000} C_DIS
LIN {X 66.010,Y 102.231,Z 70.629,A 180.000,B 0.000,C 180.000} C_DIS
LIN {X 66.024,Y 102.074,Z 70.624,A 180.000,B 0.000,C 180.000} C_DIS
LIN {X 66.038,Y 101.917,Z 70.620,A 180.000,B 0.000,C 180.000} C_DIS
LIN {X 66.045,Y 101.759,Z 70.615,A 180.000,B 0.000,C 180.000} C_DIS
LIN {X 66.045,Y 101.602,Z 70.611,A 180.000,B 0.000,C 180.000} C_DIS
LIN {X 66.045,Y 101.444,Z 70.606,A 180.000,B 0.000,C 180.000} C_DIS
LIN {X 66.045,Y 101.287,Z 70.602,A 180.000,B 0.000,C 180.000} C_DIS
LIN {X 66.041,Y 101.130,Z 70.597,A 180.000,B 0.000,C 180.000} C_DIS
LIN {X 66.028,Y 100.973,Z 70.593,A 180.000,B 0.000,C 180.000} C_DIS
LIN {X 66.014,Y 100.816,Z 70.589,A 180.000,B 0.000,C 180.000} C_DIS
LIN {X 66.000,Y 100.659,Z 70.585,A 180.000,B 0.000,C 180.000} C_DIS
LIN {X 65.984,Y 100.502,Z 70.581,A 180.000,B 0.000,C 180.000} C_DIS
LIN {X 65.959,Y 100.347,Z 70.577,A 180.000,B 0.000,C 180.000} C_DIS
LIN {X 65.931,Y 100.192,Z 70.573,A 180.000,B 0.000,C 180.000} C_DIS
